// TIA Portal project "Banda_Asamblare" (V15.1)

(* hardware
DEVICE "S71500/ET200MP station_1"  S7-1500 station
   slot 0: "Rail_0"  Rack  6ES7 590-1***0-0AA0
   slot 1: "PLC_1"  CPU 1513-1 PN  6ES7 513-1AL02-0AB0  V2.6
      slot 3: "CPU display_1"  6ES7591-1AA00-0AA0
DEVICE "HMI_1"  KTP900 Basic PN
   slot 0: "HMI_1"  KTP900 Basic PN  6AV2 123-2JB03-0AX0  15.1.0.0
   slot 1: "HMI_RT_1"  KTP900 Basic PN  6AV2 123-2JB03-0AX0  15.1.0.0
   slot 5: "HMI_1.IE_CP_1"  PROFINET Interface  15.0.1.0
      slot 1: "PROFINET Interface_1"  PROFINET Interface
         slot 1: "Port_1"  Port
*)

// ===== PLC "PLC_1"  CPU 1513-1 PN =====

VAR_GLOBAL   // PLC tag table "Default tag table"
   "Clock_Byte" AT %MB0 : Byte;
   "Clock_10Hz" AT %M0.0 : Bool;
   "Clock_5Hz" AT %M0.1 : Bool;
   "Clock_2.5Hz" AT %M0.2 : Bool;
   "Clock_2Hz" AT %M0.3 : Bool;
   "Clock_1.25Hz" AT %M0.4 : Bool;
   "Clock_1Hz" AT %M0.5 : Bool;
   "Clock_0.625Hz" AT %M0.6 : Bool;
   "Clock_0.5Hz" AT %M0.7 : Bool;
END_VAR

DATA_BLOCK "Banda1_Avarii"   // DB1
{ S7_Optimized_Access := 'TRUE' }
VERSION : 0.1
   VAR
      avarie_start : Bool;
      avarie_cuptor : Bool;
      avarie_aplatizor : Bool;
      avarie_forme : Bool;
      avarie_taiere : Bool;
      avarie_curatare : Bool;
   END_VAR
BEGIN
END_DATA_BLOCK

DATA_BLOCK "Banda1_Butoane"   // DB2
{ S7_Optimized_Access := 'TRUE' }
VERSION : 0.1
   VAR
      btn_stop : Bool;
      btn_start : Bool;
      "reset avarii" : Bool;
   END_VAR
BEGIN
END_DATA_BLOCK

DATA_BLOCK "Banda_Principala_Avarii"   // DB3
{ S7_Optimized_Access := 'TRUE' }
VERSION : 0.1
   VAR
      esd : Bool;
      btn_esd : Bool;
      reset_est : Bool;
      btn_reset_avarii : Bool;
      avarii_generale : Bool;
      avarie_piesa1 : Bool;
      avarie_piesa2 : Bool;
      avarie_piesa3 : Bool;
   END_VAR
BEGIN
END_DATA_BLOCK

DATA_BLOCK "Banda1_Mecanisme"   // DB4
{ S7_Optimized_Access := 'TRUE' }
VERSION : 0.1
   VAR
      cuptor : Bool;
      temperatura_cuptor : Real;
      "temperatura dorita la cuptor" : Real;
      aplatizor : Bool;
      forma : UInt;
      ajuns_la_forma1 : Bool;
      ajuns_la_forma2 : Bool;
      ajuns_la_forma3 : Bool;
      taiere1 : Bool;
      taiere2 : Bool;
      taiere3 : Bool;
      curatare1 : Bool;
      curatare2 : Bool;
      curatare3 : Bool;
   END_VAR
BEGIN
END_DATA_BLOCK

DATA_BLOCK "Banda2_Butoane"   // DB5
{ S7_Optimized_Access := 'TRUE' }
VERSION : 0.1
   VAR
      btn_stop : Bool;
      btn_start : Bool;
      "reset avarii" : Bool;
   END_VAR
BEGIN
END_DATA_BLOCK

DATA_BLOCK "Banda1_DB"   // DB6
{ S7_Optimized_Access := 'TRUE' }
VERSION : 0.1
// stored: InstanceOfName Banda1
"Banda1"
BEGIN
END_DATA_BLOCK

DATA_BLOCK "Banda3_DB"   // DB7
{ S7_Optimized_Access := 'TRUE' }
VERSION : 0.1
// stored: InstanceOfName Banda1
"Banda1"
BEGIN
END_DATA_BLOCK

DATA_BLOCK "Banda2_DB"   // DB8
{ S7_Optimized_Access := 'TRUE' }
VERSION : 0.1
// stored: InstanceOfName Banda1
"Banda1"
BEGIN
END_DATA_BLOCK

DATA_BLOCK "Banda1_Alarme"   // DB9
{ S7_Optimized_Access := 'TRUE' }
VERSION : 0.1
   VAR
      alarme_gather : Word;
      alarme_vect : Array[0..15] of Bool;
   END_VAR
BEGIN
END_DATA_BLOCK

DATA_BLOCK "Banda2_Alarme"   // DB11
{ S7_Optimized_Access := 'TRUE' }
VERSION : 0.1
   VAR
      alarme_gather : Word;
      alarme_vect : Array[0..15] of Bool;
   END_VAR
BEGIN
END_DATA_BLOCK

DATA_BLOCK "Banda3_Alarme"   // DB12
{ S7_Optimized_Access := 'TRUE' }
VERSION : 0.1
   VAR
      alarme_gather : Word;
      alarme_vect : Array[0..15] of Bool;
   END_VAR
BEGIN
END_DATA_BLOCK

DATA_BLOCK "Banda2_Avarii"   // DB14
{ S7_Optimized_Access := 'TRUE' }
VERSION : 0.1
   VAR
      avarie_start : Bool;
      avarie_cuptor : Bool;
      avarie_aplatizor : Bool;
      avarie_forme : Bool;
      avarie_taiere : Bool;
      avarie_curatare : Bool;
   END_VAR
BEGIN
END_DATA_BLOCK

DATA_BLOCK "Banda3_Avarii"   // DB15
{ S7_Optimized_Access := 'TRUE' }
VERSION : 0.1
   VAR
      avarie_start : Bool;
      avarie_cuptor : Bool;
      avarie_aplatizor : Bool;
      avarie_forme : Bool;
      avarie_taiere : Bool;
      avarie_curatare : Bool;
   END_VAR
BEGIN
END_DATA_BLOCK

DATA_BLOCK "Containere"   // DB16
{ S7_Optimized_Access := 'TRUE' }
VERSION : 0.1
   VAR
      container1_plin : Bool;
      container2_plin : Bool;
      container3_plin : Bool;
      container_plin_general : Bool;
      limite_containere : Bool;
      golire_c1 : Bool;
      golire_c2 : Bool;
      golire_c3 : Bool;
      container_f1 : UInt;
      container_f2 : UInt;
      container_f3 : UInt;
      limita_c1 : UInt;
      limita_c2 : UInt;
      limita_c3 : UInt;
      container_plin : Bool;
      c1_plin : Bool;
      c2_plin : Bool;
      c3_plin : Bool;
      container_final : UInt;
      limita_container_final : UInt;
      cf_plin : Bool;
      golire_cf : Bool;
      container_f1_b1 : UInt;
      container_f1_b2 : UInt;
      container_f1_b3 : UInt;
      container_f2_b1 : UInt;
      container_f2_b2 : UInt;
      container_f2_b3 : UInt;
      container_f3_b1 : UInt;
      container_f3_b2 : UInt;
      container_f3_b3 : UInt;
      container_final_1 : UInt;
      container_final_2 : UInt;
      container_final_3 : UInt;
   END_VAR
BEGIN
END_DATA_BLOCK

DATA_BLOCK "Banda3_Butoane"   // DB17
{ S7_Optimized_Access := 'TRUE' }
VERSION : 0.1
   VAR
      btn_stop : Bool;
      btn_start : Bool;
      "reset avarii" : Bool;
   END_VAR
BEGIN
END_DATA_BLOCK

DATA_BLOCK "Banda2_Mecanisme"   // DB18
{ S7_Optimized_Access := 'TRUE' }
VERSION : 0.1
   VAR
      cuptor : Bool;
      temperatura_cuptor : Real;
      "temperatura dorita la cuptor" : Real;
      aplatizor : Bool;
      forma : UInt;
      ajuns_la_forma1 : Bool;
      ajuns_la_forma2 : Bool;
      ajuns_la_forma3 : Bool;
      taiere1 : Bool;
      taiere2 : Bool;
      taiere3 : Bool;
      curatare1 : Bool;
      curatare2 : Bool;
      curatare3 : Bool;
   END_VAR
BEGIN
END_DATA_BLOCK

DATA_BLOCK "Banda3_Mecanisme"   // DB19
{ S7_Optimized_Access := 'TRUE' }
VERSION : 0.1
   VAR
      cuptor : Bool;
      temperatura_cuptor : Real;
      "temperatura dorita la cuptor" : Real;
      aplatizor : Bool;
      forma : UInt;
      ajuns_la_forma1 : Bool;
      ajuns_la_forma2 : Bool;
      ajuns_la_forma3 : Bool;
      taiere1 : Bool;
      taiere2 : Bool;
      taiere3 : Bool;
      curatare1 : Bool;
      curatare2 : Bool;
      curatare3 : Bool;
   END_VAR
BEGIN
END_DATA_BLOCK

DATA_BLOCK "Banda_Principala_Alarme"   // DB20
{ S7_Optimized_Access := 'TRUE' }
VERSION : 0.1
   VAR
      alarme_gather : Word;
      alarme_vector : Array[0..15] of Bool;
   END_VAR
BEGIN
END_DATA_BLOCK

DATA_BLOCK "Containere_Alarme"   // DB24
{ S7_Optimized_Access := 'TRUE' }
VERSION : 0.1
   VAR
      alarme_gather : Word;
      alarme_vector : Array[0..15] of Bool;
   END_VAR
BEGIN
END_DATA_BLOCK

DATA_BLOCK "Banda_Principala_Butoane"   // DB25
{ S7_Optimized_Access := 'TRUE' }
VERSION : 0.1
   VAR
      start_btn : Bool;
      stop_btn : Bool;
      pornire : Bool;
      pune_1 : Bool;
      pune_2 : Bool;
      pune_3 : Bool;
      trece_1 : Bool;
      trece_2 : Bool;
      trece_3 : Bool;
      resetare : Bool;
   END_VAR
BEGIN
END_DATA_BLOCK

DATA_BLOCK "Banda_Principala_Comenzi_DB"   // DB28
{ S7_Optimized_Access := 'TRUE' }
VERSION : 0.1
// stored: InstanceOfName Banda_Principala_Comenzi
"Banda_Principala_Comenzi"
BEGIN
END_DATA_BLOCK

DATA_BLOCK "Banda_Principala_Simulare_DB"   // DB29
{ S7_Optimized_Access := 'TRUE' }
VERSION : 0.1
// stored: InstanceOfName Banda_Principala_Simulare
"Banda_Principala_Simulare"
BEGIN
END_DATA_BLOCK

// folder: System blocks/Program resources

DATA_BLOCK "reset_buton_oprite_banda_principala"   // DB10
{ S7_Optimized_Access := 'TRUE' }
AUTHOR : Simatic
FAMILY : IEC
NAME : IEC_TMR
VERSION : 1.0
// stored: InstanceOfName IEC_TIMER
"IEC_TIMER"
BEGIN
END_DATA_BLOCK

DATA_BLOCK "reset_esd_timer"   // DB26
{ S7_Optimized_Access := 'TRUE' }
AUTHOR : Simatic
FAMILY : IEC
NAME : IEC_TMR
VERSION : 1.0
// stored: InstanceOfName IEC_TIMER
"IEC_TIMER"
BEGIN
END_DATA_BLOCK

// folder: (top level)

FUNCTION_BLOCK "Simulare1"   // FB1, LAD
{ S7_Optimized_Access := 'TRUE' }
VERSION : 0.1
   VAR_INPUT
      btn_pornire : Bool;
      b1_plecat : Bool;
      b2_plecat : Bool;
      b3_plecat : Bool;
      b41_plecat : Bool;
      b42_plecat : Bool;
      b43_plecat : Bool;
      b51_plecat : Bool;
      b52_plecat : Bool;
      b53_plecat : Bool;
      b61_plecat : Bool;
      b62_plecat : Bool;
      b63_plecat : Bool;
      cond_cuptor : Bool;
      forma : UInt;
      trecere_banda_mare1 : Bool;
      trecere_banda_mare2 : Bool;
      trecere_banda_mare3 : Bool;
   END_VAR
   VAR_OUTPUT
      cuptor_pornit : Bool;
      aplatizor_pornit : Bool;
      forma1 : Bool;
      forma2 : Bool;
      forma3 : Bool;
      taiere1 : Bool;
      taiere2 : Bool;
      taiere3 : Bool;
      curatare1 : Bool;
      curatare2 : Bool;
      curatare3 : Bool;
      container1 : UInt;
      container2 : UInt;
      container3 : UInt;
      servo : UInt;
   END_VAR
   VAR_IN_OUT
      pune_material : Bool;
      temp_cuptor : Real;
      golire_c1 : Bool;
      golire_c2 : Bool;
      golire_c3 : Bool;
   END_VAR
   VAR
      re1 : Bool;
      re2 : Bool;
      re3 : Bool;
      re4 : Bool;
      re5 : Bool;
      re6 : Bool;
      re7 : Bool;
      re8 : Bool;
      "timer reset punere material" : TON_TIME;
      mentinere_timer_material : Bool;
      timer_aplatizare : TON_TIME;
      "tiimer forma" : TON_TIME;
      "timer taiere1" : TON_TIME;
      "timer taiere2" : TON_TIME;
      "timer taiere3" : TON_TIME;
      "timer curatare1" : TON_TIME;
      "timer curatare 2" : TON_TIME;
      "timer curatare 3" : TON_TIME;
      reset_golire1 : TON_TIME;
      reset_golire2 : TON_TIME;
      reset_golire3 : TON_TIME;
      scazut1 : Bool;
      scazut2 : Bool;
      scazut3 : Bool;
   END_VAR
   VAR_TEMP   // added for the SCL form of the ladder/FBD networks
      _w1 : Bool;
      _w2 : Bool;
      _w3 : Bool;
   END_VAR
BEGIN

REGION Network 1: pune un block de material pe banda
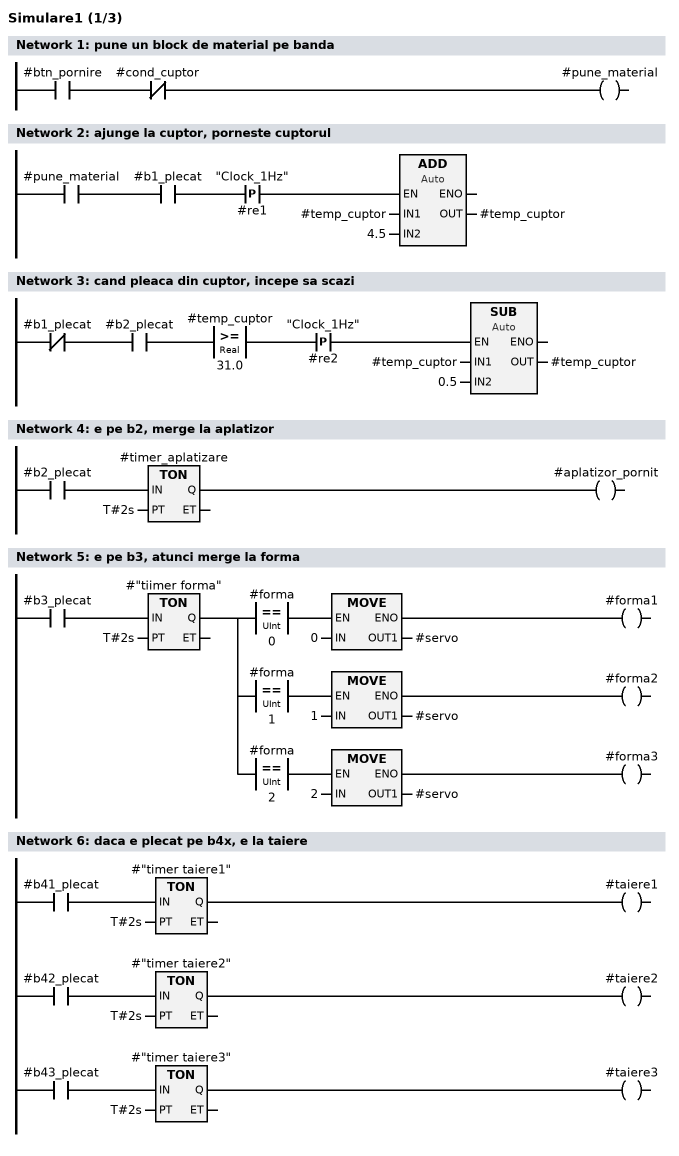
   RUNG wire#powerrail
      Contact( #btn_pornire )
      I_Contact( #cond_cuptor )
      Coil( #pune_material )
   END_RUNG
   // the same network as SCL:
   #pune_material := #btn_pornire AND NOT #cond_cuptor;
END_REGION

REGION Network 2: ajunge la cuptor, porneste cuptorul
   RUNG wire#powerrail
      Contact( #pune_material )
      Contact( #b1_plecat )
      P_Contact(operand := "Clock_1Hz", bit := #re1)
      Add(in1 := #temp_cuptor, in2 := 4.5, out => #temp_cuptor)
   END_RUNG
   // the same network as SCL:
   #_w1 := #pune_material AND #b1_plecat AND "Clock_1Hz" AND NOT #re1;   // rising edge of "Clock_1Hz"
   #re1 := "Clock_1Hz";
   IF #_w1 THEN #temp_cuptor := #temp_cuptor + 4.5; END_IF;
END_REGION

REGION Network 3: cand pleaca din cuptor, incepe sa scazi
   RUNG wire#powerrail
      I_Contact( #b1_plecat )
      Contact( #b2_plecat )
      { S7_Templates := "SrcType := Real" } GE_Contact(in1 := #temp_cuptor, in2 := 31.0)
      P_Contact(operand := "Clock_1Hz", bit := #re2)
      Sub(in1 := #temp_cuptor, in2 := 0.5, out => #temp_cuptor)
   END_RUNG
   // the same network as SCL:
   #_w1 := NOT #b1_plecat AND #b2_plecat AND (#temp_cuptor >= 31.0) AND "Clock_1Hz" AND NOT #re2;   // rising edge of "Clock_1Hz"
   #re2 := "Clock_1Hz";
   IF #_w1 THEN #temp_cuptor := #temp_cuptor - 0.5; END_IF;
END_REGION

REGION Network 4: e pe b2, merge la aplatizor
   #timer_aplatizare(IN := #b2_plecat, PT := T#2s);   // TON
   #aplatizor_pornit := #timer_aplatizare.Q;
END_REGION

REGION Network 5: e pe b3, atunci merge la forma
   #"tiimer forma"(IN := #b3_plecat, PT := T#2s);   // TON
   #_w1 := #"tiimer forma".Q AND (#forma = 0);
   IF #_w1 THEN #servo := 0; END_IF;
   #forma1 := #_w1;
   #_w2 := #"tiimer forma".Q AND (#forma = 1);
   IF #_w2 THEN #servo := 1; END_IF;
   #forma2 := #_w2;
   #_w3 := #"tiimer forma".Q AND (#forma = 2);
   IF #_w3 THEN #servo := 2; END_IF;
   #forma3 := #_w3;
END_REGION

REGION Network 6: daca e plecat pe b4x, e la taiere
   #"timer taiere1"(IN := #b41_plecat, PT := T#2s);   // TON
   #taiere1 := #"timer taiere1".Q;
   #"timer taiere2"(IN := #b42_plecat, PT := T#2s);   // TON
   #taiere2 := #"timer taiere2".Q;
   #"timer taiere3"(IN := #b43_plecat, PT := T#2s);   // TON
   #taiere3 := #"timer taiere3".Q;
END_REGION

REGION Network 7: daca e pe banda b5x, sa dea drumul la curatari
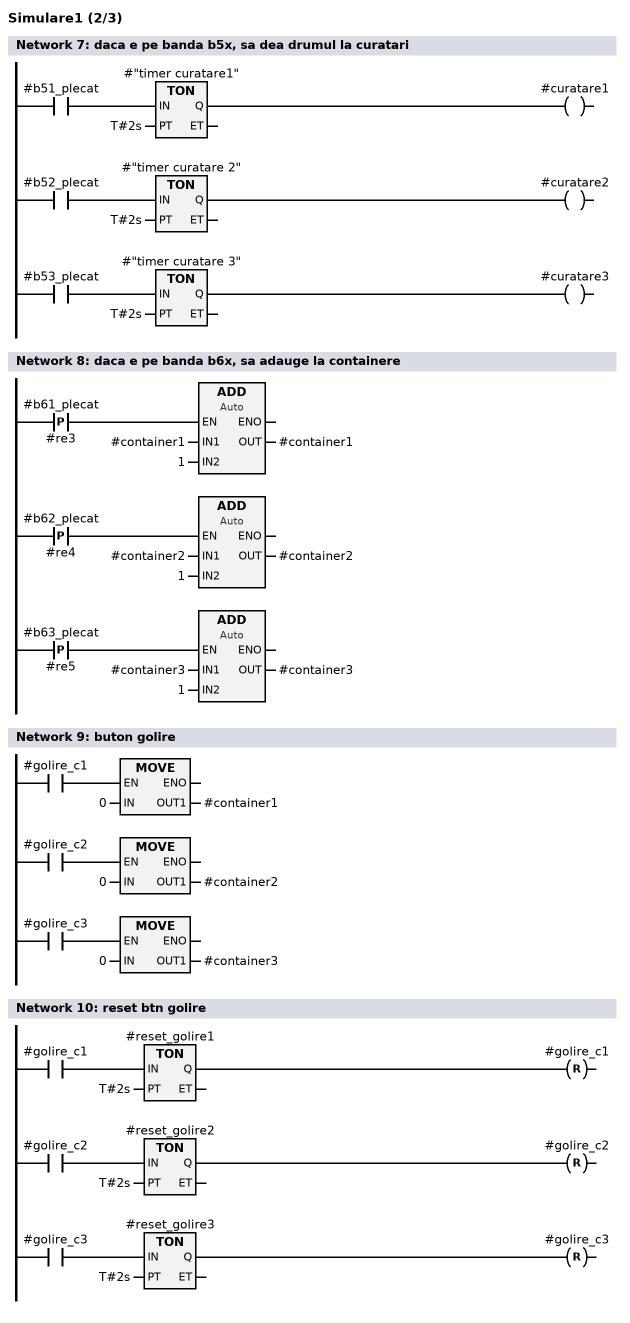
   #"timer curatare1"(IN := #b51_plecat, PT := T#2s);   // TON
   #curatare1 := #"timer curatare1".Q;
   #"timer curatare 2"(IN := #b52_plecat, PT := T#2s);   // TON
   #curatare2 := #"timer curatare 2".Q;
   #"timer curatare 3"(IN := #b53_plecat, PT := T#2s);   // TON
   #curatare3 := #"timer curatare 3".Q;
END_REGION

REGION Network 8: daca e pe banda b6x, sa adauge la containere
   RUNG wire#powerrail
      P_Contact(operand := #b61_plecat, bit := #re3)
      Add(in1 := #container1, in2 := 1, out => #container1)
   END_RUNG
   RUNG wire#powerrail
      P_Contact(operand := #b62_plecat, bit := #re4)
      Add(in1 := #container2, in2 := 1, out => #container2)
   END_RUNG
   RUNG wire#powerrail
      P_Contact(operand := #b63_plecat, bit := #re5)
      Add(in1 := #container3, in2 := 1, out => #container3)
   END_RUNG
   // the same network as SCL:
   #_w1 := #b61_plecat AND NOT #re3;   // rising edge of #b61_plecat
   #re3 := #b61_plecat;
   IF #_w1 THEN #container1 := #container1 + 1; END_IF;
   #_w2 := #b62_plecat AND NOT #re4;   // rising edge of #b62_plecat
   #re4 := #b62_plecat;
   IF #_w2 THEN #container2 := #container2 + 1; END_IF;
   #_w3 := #b63_plecat AND NOT #re5;   // rising edge of #b63_plecat
   #re5 := #b63_plecat;
   IF #_w3 THEN #container3 := #container3 + 1; END_IF;
END_REGION

REGION Network 9: buton golire
   RUNG wire#powerrail
      Contact( #golire_c1 )
      Move(in := 0, out1 => #container1)
   END_RUNG
   RUNG wire#powerrail
      Contact( #golire_c2 )
      Move(in := 0, out1 => #container2)
   END_RUNG
   RUNG wire#powerrail
      Contact( #golire_c3 )
      Move(in := 0, out1 => #container3)
   END_RUNG
   // the same network as SCL:
   IF #golire_c1 THEN #container1 := 0; END_IF;
   IF #golire_c2 THEN #container2 := 0; END_IF;
   IF #golire_c3 THEN #container3 := 0; END_IF;
END_REGION

REGION Network 10: reset btn golire
   #reset_golire1(IN := #golire_c1, PT := T#2s);   // TON
   IF #reset_golire1.Q THEN #golire_c1 := FALSE; END_IF;
   #reset_golire2(IN := #golire_c2, PT := T#2s);   // TON
   IF #reset_golire2.Q THEN #golire_c2 := FALSE; END_IF;
   #reset_golire3(IN := #golire_c3, PT := T#2s);   // TON
   IF #reset_golire3.Q THEN #golire_c3 := FALSE; END_IF;
END_REGION

REGION Network 11: daca avem treceri de pe banda mare, scadem valoarea din containere
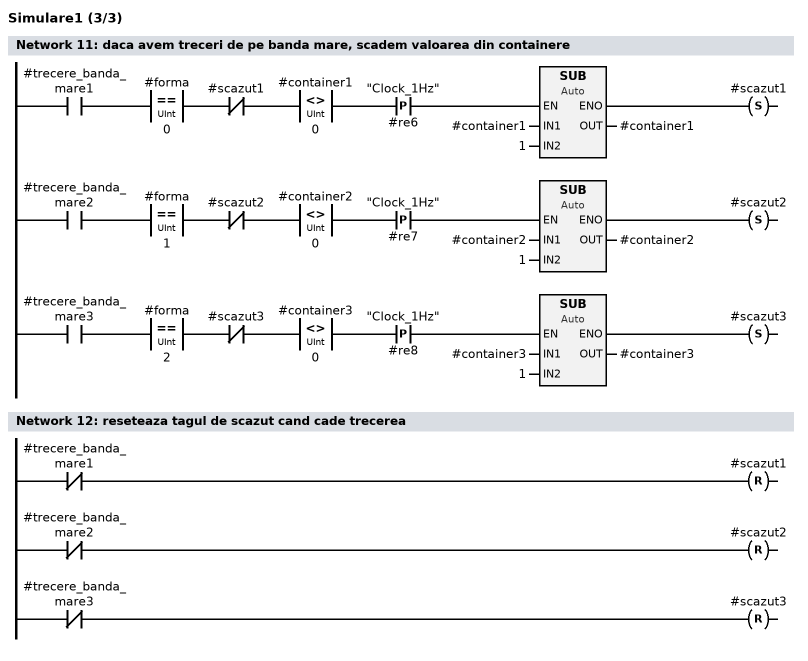
   RUNG wire#powerrail
      Contact( #trecere_banda_mare1 )
      { S7_Templates := "SrcType := UInt" } EQ_Contact(in1 := #forma, in2 := 0)
      I_Contact( #scazut1 )
      { S7_Templates := "SrcType := UInt" } NE_Contact(in1 := #container1, in2 := 0)
      P_Contact(operand := "Clock_1Hz", bit := #re6)
      Sub(in1 := #container1, in2 := 1, out => #container1)
      S_Coil( #scazut1 )
   END_RUNG
   RUNG wire#powerrail
      Contact( #trecere_banda_mare2 )
      { S7_Templates := "SrcType := UInt" } EQ_Contact(in1 := #forma, in2 := 1)
      I_Contact( #scazut2 )
      { S7_Templates := "SrcType := UInt" } NE_Contact(in1 := #container2, in2 := 0)
      P_Contact(operand := "Clock_1Hz", bit := #re7)
      Sub(in1 := #container2, in2 := 1, out => #container2)
      S_Coil( #scazut2 )
   END_RUNG
   RUNG wire#powerrail
      Contact( #trecere_banda_mare3 )
      { S7_Templates := "SrcType := UInt" } EQ_Contact(in1 := #forma, in2 := 2)
      I_Contact( #scazut3 )
      { S7_Templates := "SrcType := UInt" } NE_Contact(in1 := #container3, in2 := 0)
      P_Contact(operand := "Clock_1Hz", bit := #re8)
      Sub(in1 := #container3, in2 := 1, out => #container3)
      S_Coil( #scazut3 )
   END_RUNG
   // the same network as SCL:
   #_w1 := #trecere_banda_mare1 AND (#forma = 0) AND NOT #scazut1 AND (#container1 <> 0) AND "Clock_1Hz" AND NOT #re6;   // rising edge of "Clock_1Hz"
   #re6 := "Clock_1Hz";
   IF #_w1 THEN
       #container1 := #container1 - 1;
       #scazut1 := TRUE;
   END_IF;
   #_w2 := #trecere_banda_mare2 AND (#forma = 1) AND NOT #scazut2 AND (#container2 <> 0) AND "Clock_1Hz" AND NOT #re7;   // rising edge of "Clock_1Hz"
   #re7 := "Clock_1Hz";
   IF #_w2 THEN
       #container2 := #container2 - 1;
       #scazut2 := TRUE;
   END_IF;
   #_w3 := #trecere_banda_mare3 AND (#forma = 2) AND NOT #scazut3 AND (#container3 <> 0) AND "Clock_1Hz" AND NOT #re8;   // rising edge of "Clock_1Hz"
   #re8 := "Clock_1Hz";
   IF #_w3 THEN
       #container3 := #container3 - 1;
       #scazut3 := TRUE;
   END_IF;
END_REGION

REGION Network 12: reseteaza tagul de scazut cand cade trecerea
   RUNG wire#powerrail
      I_Contact( #trecere_banda_mare1 )
      R_Coil( #scazut1 )
   END_RUNG
   RUNG wire#powerrail
      I_Contact( #trecere_banda_mare2 )
      R_Coil( #scazut2 )
   END_RUNG
   RUNG wire#powerrail
      I_Contact( #trecere_banda_mare3 )
      R_Coil( #scazut3 )
   END_RUNG
   // the same network as SCL:
   IF NOT #trecere_banda_mare1 THEN #scazut1 := FALSE; END_IF;
   IF NOT #trecere_banda_mare2 THEN #scazut2 := FALSE; END_IF;
   IF NOT #trecere_banda_mare3 THEN #scazut3 := FALSE; END_IF;
END_REGION
END_FUNCTION_BLOCK

FUNCTION_BLOCK "Comenzi1"   // FB2, LAD
{ S7_Optimized_Access := 'TRUE' }
VERSION : 0.1
   VAR_INPUT
      temp_cuptor : Real;
      temp_dorita : Real;
      pune_material : Bool;
      aplatizor_pornit : Bool;
      forma1 : Bool;
      forma2 : Bool;
      forma3 : Bool;
      taiere1 : Bool;
      taiere2 : Bool;
      taiere3 : Bool;
      curatare1 : Bool;
      curatare2 : Bool;
      curatare3 : Bool;
   END_VAR
   VAR_OUTPUT
      b1_plecat : Bool;
      b2_plecat : Bool;
      b3_plecat : Bool;
      b41_plecat : Bool;
      b42_plecat : Bool;
      b43_plecat : Bool;
      b51_plecat : Bool;
      b52_plecat : Bool;
      b53_plecat : Bool;
      b61_plecat : Bool;
      b62_plecat : Bool;
      b63_plecat : Bool;
      cond_cuptor : Bool;
   END_VAR
   VAR
      "timer plecare b1" : TON_TIME;
      incc : Int;
      edg : Bool;
   END_VAR
BEGIN

REGION Network 1: pleaca spre cuptor
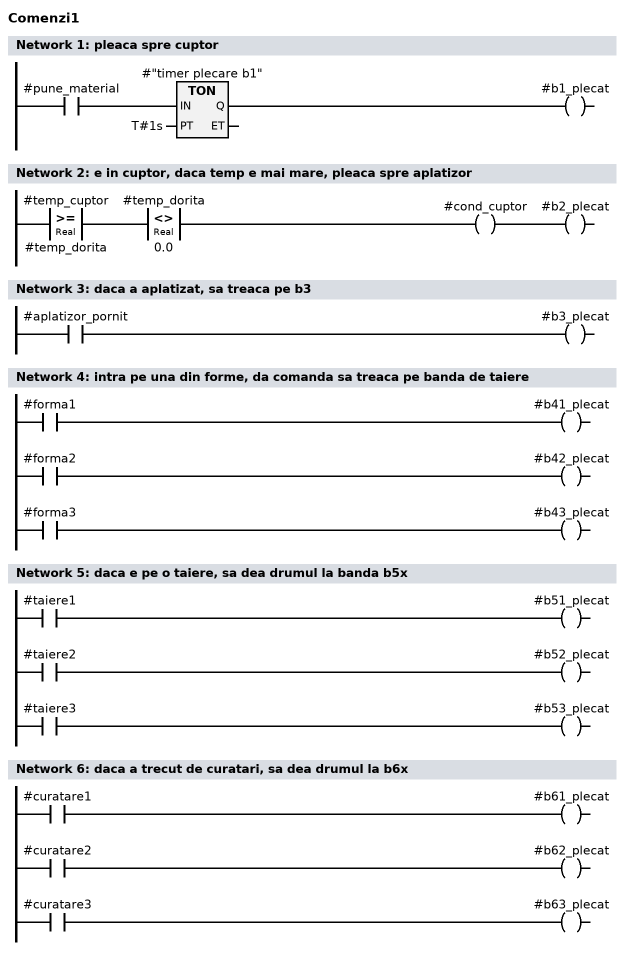
   #"timer plecare b1"(IN := #pune_material, PT := T#1s);   // TON
   #b1_plecat := #"timer plecare b1".Q;
END_REGION

REGION Network 2: e in cuptor, daca temp e mai mare, pleaca spre aplatizor
   RUNG wire#powerrail
      { S7_Templates := "SrcType := Real" } GE_Contact(in1 := #temp_cuptor, in2 := #temp_dorita)
      { S7_Templates := "SrcType := Real" } NE_Contact(in1 := #temp_dorita, in2 := 0.0)
      Coil( #cond_cuptor )
      Coil( #b2_plecat )
   END_RUNG
   // the same network as SCL:
   #cond_cuptor := (#temp_cuptor >= #temp_dorita) AND (#temp_dorita <> 0.0);
   #b2_plecat := #cond_cuptor;
END_REGION

REGION Network 3: daca a aplatizat, sa treaca pe b3
   RUNG wire#powerrail
      Contact( #aplatizor_pornit )
      Coil( #b3_plecat )
   END_RUNG
   // the same network as SCL:
   #b3_plecat := #aplatizor_pornit;
END_REGION

REGION Network 4: intra pe una din forme, da comanda sa treaca pe banda de taiere
   RUNG wire#powerrail
      Contact( #forma1 )
      Coil( #b41_plecat )
   END_RUNG
   RUNG wire#powerrail
      Contact( #forma2 )
      Coil( #b42_plecat )
   END_RUNG
   RUNG wire#powerrail
      Contact( #forma3 )
      Coil( #b43_plecat )
   END_RUNG
   // the same network as SCL:
   #b41_plecat := #forma1;
   #b42_plecat := #forma2;
   #b43_plecat := #forma3;
END_REGION

REGION Network 5: daca e pe o taiere, sa dea drumul la banda b5x
   RUNG wire#powerrail
      Contact( #taiere1 )
      Coil( #b51_plecat )
   END_RUNG
   RUNG wire#powerrail
      Contact( #taiere2 )
      Coil( #b52_plecat )
   END_RUNG
   RUNG wire#powerrail
      Contact( #taiere3 )
      Coil( #b53_plecat )
   END_RUNG
   // the same network as SCL:
   #b51_plecat := #taiere1;
   #b52_plecat := #taiere2;
   #b53_plecat := #taiere3;
END_REGION

REGION Network 6: daca a trecut de curatari, sa dea drumul la b6x
   RUNG wire#powerrail
      Contact( #curatare1 )
      Coil( #b61_plecat )
   END_RUNG
   RUNG wire#powerrail
      Contact( #curatare2 )
      Coil( #b62_plecat )
   END_RUNG
   RUNG wire#powerrail
      Contact( #curatare3 )
      Coil( #b63_plecat )
   END_RUNG
   // the same network as SCL:
   #b61_plecat := #curatare1;
   #b62_plecat := #curatare2;
   #b63_plecat := #curatare3;
END_REGION
END_FUNCTION_BLOCK

FUNCTION_BLOCK "Banda1"   // FB3, LAD
{ S7_Optimized_Access := 'TRUE' }
VERSION : 0.1
   VAR_INPUT
      temperatura_dorita : Real := 0.0;
      forma : UInt := 0;
      limita_container1 : UInt;
      limita_container2 : UInt;
      limita_container3 : UInt;
      container_plin : Bool;
      trecere_banda_mare1 : Bool;
      trecere_banda_mare2 : Bool;
      trecere_banda_mare3 : Bool;
   END_VAR
   VAR_OUTPUT
      container1 : UInt;
      container2 : UInt;
      container3 : UInt;
      cuptor : Bool;
      aplatizor : Bool;
      ajuns_forma1 : Bool;
      ajuns_forma2 : Bool;
      ajuns_forma3 : Bool;
      taiere1 : Bool;
      taiere2 : Bool;
      taiere3 : Bool;
      curatare1 : Bool;
      curatare2 : Bool;
      curatare3 : Bool;
      alarme_gather : Word;
      alarme_vect : Array[0..15] of Bool;
   END_VAR
   VAR_IN_OUT
      stop : Bool;
      start : Bool;
      golire_c1 : Bool;
      golire_c2 : Bool;
      golire_c3 : Bool;
      btn_reset_avarii : Bool;
      avarie_start : Bool;
      avarie_cuptor : Bool;
      avarie_aplatizor : Bool;
      avarie_forma : Bool;
      avarie_taiere : Bool;
      avarie_curatare : Bool;
      temperatura_cuptor : Real;
      esd : Bool;
   END_VAR
   VAR
      limite_containere : Bool;
      Avarii_generale : Bool;
      pornire : Bool;
      punere_block : Bool;
      plecat_b1 : Bool;
      plecat_b2 : Bool;
      plecat_b3 : Bool;
      plecat_b41 : Bool;
      plecat_b42 : Bool;
      plecat_b43 : Bool;
      plecar_b51 : Bool;
      plecar_b52 : Bool;
      plecar_b53 : Bool;
      plecat_b61 : Bool;
      plecat_b62 : Bool;
      plecat_b63 : Bool;
      cond_cuptor : Bool;
      servo : UInt;
      reset_esd_timer : TON_TIME;
      plin_container1 : Bool;
      plin_container2 : Bool;
      plin_container3 : Bool;
      reset_btn_stop : TON_TIME;
      Simulare1_Instance : "Simulare1";
      Comenzi1_Instance : "Comenzi1";
   END_VAR
BEGIN

REGION Network 1: buton start
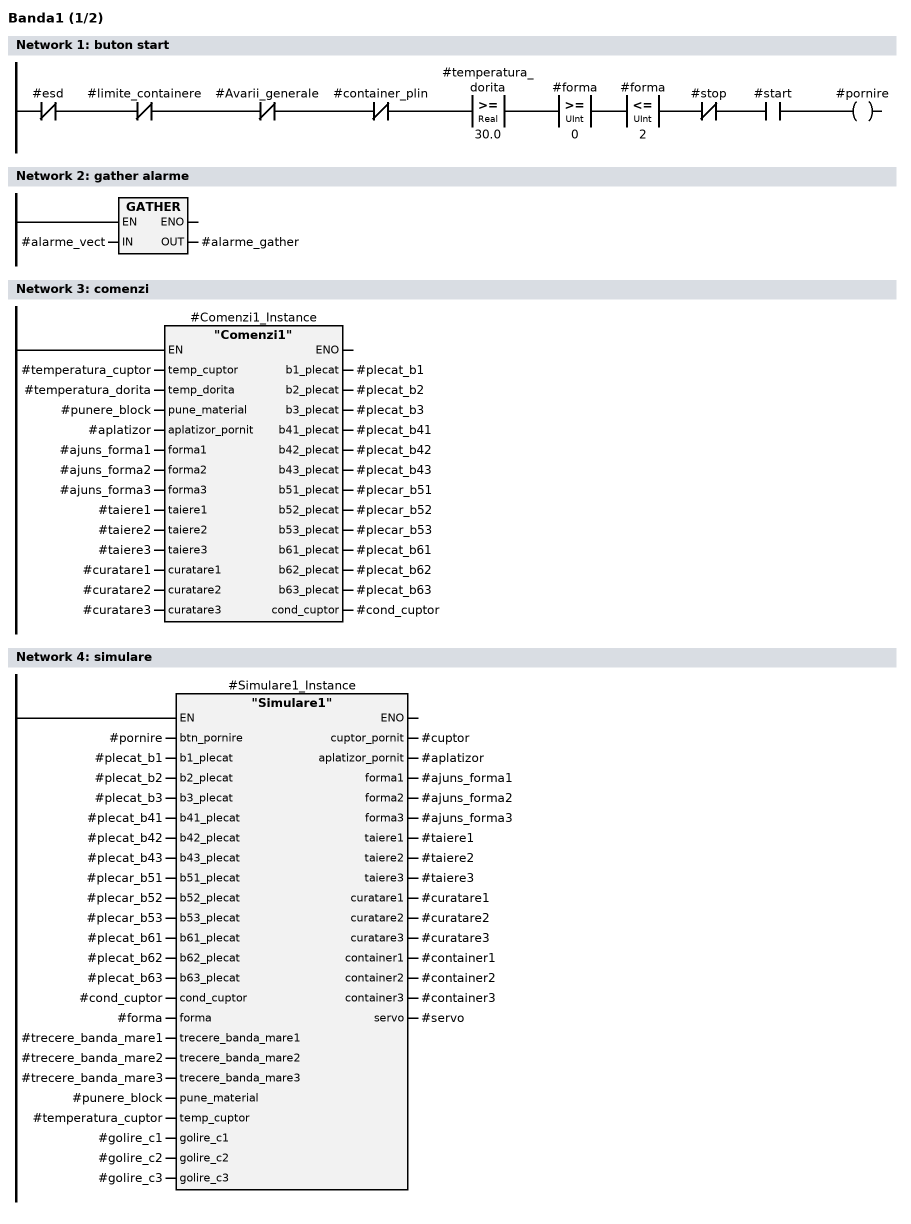
   RUNG wire#powerrail
      I_Contact( #esd )
      I_Contact( #limite_containere )
      I_Contact( #Avarii_generale )
      I_Contact( #container_plin )
      { S7_Templates := "SrcType := Real" } GE_Contact(in1 := #temperatura_dorita, in2 := 30.0)
      { S7_Templates := "SrcType := UInt" } GE_Contact(in1 := #forma, in2 := 0)
      { S7_Templates := "SrcType := UInt" } LE_Contact(in1 := #forma, in2 := 2)
      I_Contact( #stop )
      Contact( #start )
      Coil( #pornire )
   END_RUNG
   // the same network as SCL:
   #pornire := NOT #esd AND NOT #limite_containere AND NOT #Avarii_generale AND NOT #container_plin AND (#temperatura_dorita >= 30.0) AND (#forma >= 0) AND (#forma <= 2) AND NOT #stop AND #start;
END_REGION

REGION Network 2: gather alarme
   GATHER(IN := #alarme_vect, OUT => #alarme_gather);
END_REGION

REGION Network 3: comenzi
   RUNG wire#powerrail
      #Comenzi1_Instance(temp_cuptor := #temperatura_cuptor, temp_dorita := #temperatura_dorita, pune_material := #punere_block, aplatizor_pornit := #aplatizor, forma1 := #ajuns_forma1, forma2 := #ajuns_forma2, forma3 := #ajuns_forma3, taiere1 := #taiere1, taiere2 := #taiere2, taiere3 := #taiere3, curatare1 := #curatare1, curatare2 := #curatare2, curatare3 := #curatare3, b1_plecat => #plecat_b1, b2_plecat => #plecat_b2, b3_plecat => #plecat_b3, b41_plecat => #plecat_b41, b42_plecat => #plecat_b42, b43_plecat => #plecat_b43, b51_plecat => #plecar_b51, b52_plecat => #plecar_b52, b53_plecat => #plecar_b53, b61_plecat => #plecat_b61, b62_plecat => #plecat_b62, b63_plecat => #plecat_b63, cond_cuptor => #cond_cuptor)
   END_RUNG
   // the same network as SCL:
   #Comenzi1_Instance(temp_cuptor := #temperatura_cuptor,   // "Comenzi1"
                      temp_dorita := #temperatura_dorita,
                      pune_material := #punere_block,
                      aplatizor_pornit := #aplatizor,
                      forma1 := #ajuns_forma1,
                      forma2 := #ajuns_forma2,
                      forma3 := #ajuns_forma3,
                      taiere1 := #taiere1,
                      taiere2 := #taiere2,
                      taiere3 := #taiere3,
                      curatare1 := #curatare1,
                      curatare2 := #curatare2,
                      curatare3 := #curatare3,
                      b1_plecat => #plecat_b1,
                      b2_plecat => #plecat_b2,
                      b3_plecat => #plecat_b3,
                      b41_plecat => #plecat_b41,
                      b42_plecat => #plecat_b42,
                      b43_plecat => #plecat_b43,
                      b51_plecat => #plecar_b51,
                      b52_plecat => #plecar_b52,
                      b53_plecat => #plecar_b53,
                      b61_plecat => #plecat_b61,
                      b62_plecat => #plecat_b62,
                      b63_plecat => #plecat_b63,
                      cond_cuptor => #cond_cuptor);
END_REGION

REGION Network 4: simulare
   RUNG wire#powerrail
      #Simulare1_Instance(btn_pornire := #pornire, b1_plecat := #plecat_b1, b2_plecat := #plecat_b2, b3_plecat := #plecat_b3, b41_plecat := #plecat_b41, b42_plecat := #plecat_b42, b43_plecat := #plecat_b43, b51_plecat := #plecar_b51, b52_plecat := #plecar_b52, b53_plecat := #plecar_b53, b61_plecat := #plecat_b61, b62_plecat := #plecat_b62, b63_plecat := #plecat_b63, cond_cuptor := #cond_cuptor, forma := #forma, trecere_banda_mare1 := #trecere_banda_mare1, trecere_banda_mare2 := #trecere_banda_mare2, trecere_banda_mare3 := #trecere_banda_mare3, pune_material := #punere_block, temp_cuptor := #temperatura_cuptor, golire_c1 := #golire_c1, golire_c2 := #golire_c2, golire_c3 := #golire_c3, cuptor_pornit => #cuptor, aplatizor_pornit => #aplatizor, forma1 => #ajuns_forma1, forma2 => #ajuns_forma2, forma3 => #ajuns_forma3, taiere1 => #taiere1, taiere2 => #taiere2, taiere3 => #taiere3, curatare1 => #curatare1, curatare2 => #curatare2, curatare3 => #curatare3, container1 => #container1, container2 => #container2, container3 => #container3, servo => #servo)
   END_RUNG
   // the same network as SCL:
   #Simulare1_Instance(btn_pornire := #pornire,   // "Simulare1"
                       b1_plecat := #plecat_b1,
                       b2_plecat := #plecat_b2,
                       b3_plecat := #plecat_b3,
                       b41_plecat := #plecat_b41,
                       b42_plecat := #plecat_b42,
                       b43_plecat := #plecat_b43,
                       b51_plecat := #plecar_b51,
                       b52_plecat := #plecar_b52,
                       b53_plecat := #plecar_b53,
                       b61_plecat := #plecat_b61,
                       b62_plecat := #plecat_b62,
                       b63_plecat := #plecat_b63,
                       cond_cuptor := #cond_cuptor,
                       forma := #forma,
                       trecere_banda_mare1 := #trecere_banda_mare1,
                       trecere_banda_mare2 := #trecere_banda_mare2,
                       trecere_banda_mare3 := #trecere_banda_mare3,
                       pune_material := #punere_block,
                       temp_cuptor := #temperatura_cuptor,
                       golire_c1 := #golire_c1,
                       golire_c2 := #golire_c2,
                       golire_c3 := #golire_c3,
                       cuptor_pornit => #cuptor,
                       aplatizor_pornit => #aplatizor,
                       forma1 => #ajuns_forma1,
                       forma2 => #ajuns_forma2,
                       forma3 => #ajuns_forma3,
                       taiere1 => #taiere1,
                       taiere2 => #taiere2,
                       taiere3 => #taiere3,
                       curatare1 => #curatare1,
                       curatare2 => #curatare2,
                       curatare3 => #curatare3,
                       container1 => #container1,
                       container2 => #container2,
                       container3 => #container3,
                       servo => #servo);
END_REGION

REGION Network 5: avarie generala
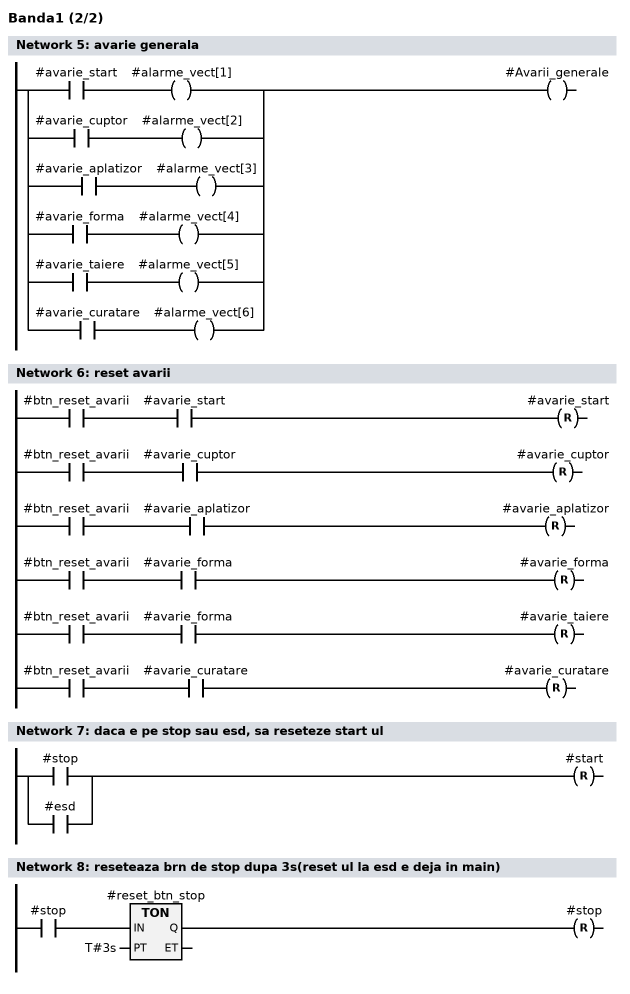
   RUNG wire#powerrail
      Contact( #avarie_start )
      Coil( #alarme_vect[1] )
      wire#w1
      Coil( #Avarii_generale )
   END_RUNG
   RUNG wire#powerrail
      Contact( #avarie_cuptor )
      Coil( #alarme_vect[2] )
   END_RUNG wire#w1
   RUNG wire#powerrail
      Contact( #avarie_aplatizor )
      Coil( #alarme_vect[3] )
   END_RUNG wire#w1
   RUNG wire#powerrail
      Contact( #avarie_forma )
      Coil( #alarme_vect[4] )
   END_RUNG wire#w1
   RUNG wire#powerrail
      Contact( #avarie_taiere )
      Coil( #alarme_vect[5] )
   END_RUNG wire#w1
   RUNG wire#powerrail
      Contact( #avarie_curatare )
      Coil( #alarme_vect[6] )
   END_RUNG wire#w1
   // the same network as SCL:
   #alarme_vect[1] := #avarie_start;
   #alarme_vect[2] := #avarie_cuptor;
   #alarme_vect[3] := #avarie_aplatizor;
   #alarme_vect[4] := #avarie_forma;
   #alarme_vect[5] := #avarie_taiere;
   #alarme_vect[6] := #avarie_curatare;
   #Avarii_generale := #avarie_start OR #avarie_cuptor OR #avarie_aplatizor OR #avarie_forma OR #avarie_taiere OR #avarie_curatare;
END_REGION

REGION Network 6: reset avarii
   RUNG wire#powerrail
      Contact( #btn_reset_avarii )
      Contact( #avarie_start )
      R_Coil( #avarie_start )
   END_RUNG
   RUNG wire#powerrail
      Contact( #btn_reset_avarii )
      Contact( #avarie_cuptor )
      R_Coil( #avarie_cuptor )
   END_RUNG
   RUNG wire#powerrail
      Contact( #btn_reset_avarii )
      Contact( #avarie_aplatizor )
      R_Coil( #avarie_aplatizor )
   END_RUNG
   RUNG wire#powerrail
      Contact( #btn_reset_avarii )
      Contact( #avarie_forma )
      R_Coil( #avarie_forma )
   END_RUNG
   RUNG wire#powerrail
      Contact( #btn_reset_avarii )
      Contact( #avarie_forma )
      R_Coil( #avarie_taiere )
   END_RUNG
   RUNG wire#powerrail
      Contact( #btn_reset_avarii )
      Contact( #avarie_curatare )
      R_Coil( #avarie_curatare )
   END_RUNG
   // the same network as SCL:
   IF #btn_reset_avarii AND #avarie_start THEN #avarie_start := FALSE; END_IF;
   IF #btn_reset_avarii AND #avarie_cuptor THEN #avarie_cuptor := FALSE; END_IF;
   IF #btn_reset_avarii AND #avarie_aplatizor THEN #avarie_aplatizor := FALSE; END_IF;
   IF #btn_reset_avarii AND #avarie_forma THEN #avarie_forma := FALSE; END_IF;
   IF #btn_reset_avarii AND #avarie_forma THEN #avarie_taiere := FALSE; END_IF;
   IF #btn_reset_avarii AND #avarie_curatare THEN #avarie_curatare := FALSE; END_IF;
END_REGION

REGION Network 7: daca e pe stop sau esd, sa reseteze start ul
   RUNG wire#powerrail
      Contact( #stop )
      wire#w1
      R_Coil( #start )
   END_RUNG
   RUNG wire#powerrail
      Contact( #esd )
   END_RUNG wire#w1
   // the same network as SCL:
   IF #stop OR #esd THEN #start := FALSE; END_IF;
END_REGION

REGION Network 8: reseteaza brn de stop dupa 3s(reset ul la esd e deja in main)
   #reset_btn_stop(IN := #stop, PT := T#3s);   // TON
   IF #reset_btn_stop.Q THEN #stop := FALSE; END_IF;
END_REGION
END_FUNCTION_BLOCK

FUNCTION_BLOCK "Banda_Principala_Comenzi"   // FB4, LAD
{ S7_Optimized_Access := 'TRUE' }
VERSION : 0.1
   VAR_INPUT
      pornire : Bool;
      trecut1 : Bool;
      trecut2 : Bool;
      resetare : Bool;
   END_VAR
   VAR_OUTPUT
      pune_1 : Bool;
      pune_2 : Bool;
      pune_3 : Bool;
   END_VAR
BEGIN

REGION Network 1: daca e pornit, pune pentru forma1
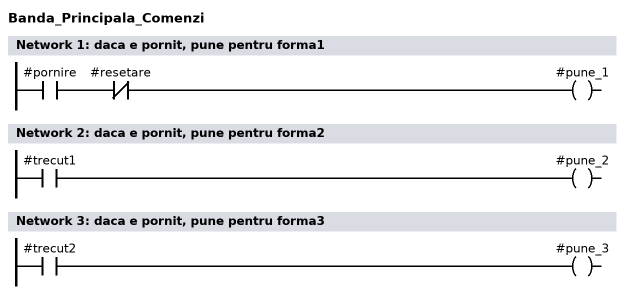
   RUNG wire#powerrail
      Contact( #pornire )
      I_Contact( #resetare )
      Coil( #pune_1 )
   END_RUNG
   // the same network as SCL:
   #pune_1 := #pornire AND NOT #resetare;
END_REGION

REGION Network 2: daca e pornit, pune pentru forma2
   RUNG wire#powerrail
      Contact( #trecut1 )
      Coil( #pune_2 )
   END_RUNG
   // the same network as SCL:
   #pune_2 := #trecut1;
END_REGION

REGION Network 3: daca e pornit, pune pentru forma3
   RUNG wire#powerrail
      Contact( #trecut2 )
      Coil( #pune_3 )
   END_RUNG
   // the same network as SCL:
   #pune_3 := #trecut2;
END_REGION
END_FUNCTION_BLOCK

FUNCTION_BLOCK "Banda_Principala_Simulare"   // FB5, LAD
{ S7_Optimized_Access := 'TRUE' }
VERSION : 0.1
   VAR_INPUT
      pune1 : Bool;
      pune2 : Bool;
      pune3 : Bool;
   END_VAR
   VAR_OUTPUT
      container_final : UInt;
      container_final_1 : UInt;
      container_final_2 : UInt;
      container_final_3 : UInt;
      trecut1 : Bool;
      trecut2 : Bool;
      trecut3 : Bool;
      resetare : Bool;
      alarma1 : Bool;
      alarma2 : Bool;
      alarma3 : Bool;
   END_VAR
   VAR_IN_OUT
      container1 : UInt;
      container2 : UInt;
      container3 : UInt;
      golire_container_final : Bool;
   END_VAR
   VAR
      timer_f1 : TON_TIME;
      timer_f2 : TON_TIME;
      timer_f3 : TON_TIME;
      re1 : Bool;
      reset_btn_golire : TON_TIME;
      timer_resetare : TON_TIME;
   END_VAR
   VAR_TEMP   // added for the SCL form of the ladder/FBD networks
      _w1 : Bool;
   END_VAR
BEGIN

REGION Network 1: daca poate pune pe 1, si containerulnu e pe 0, pune si continua
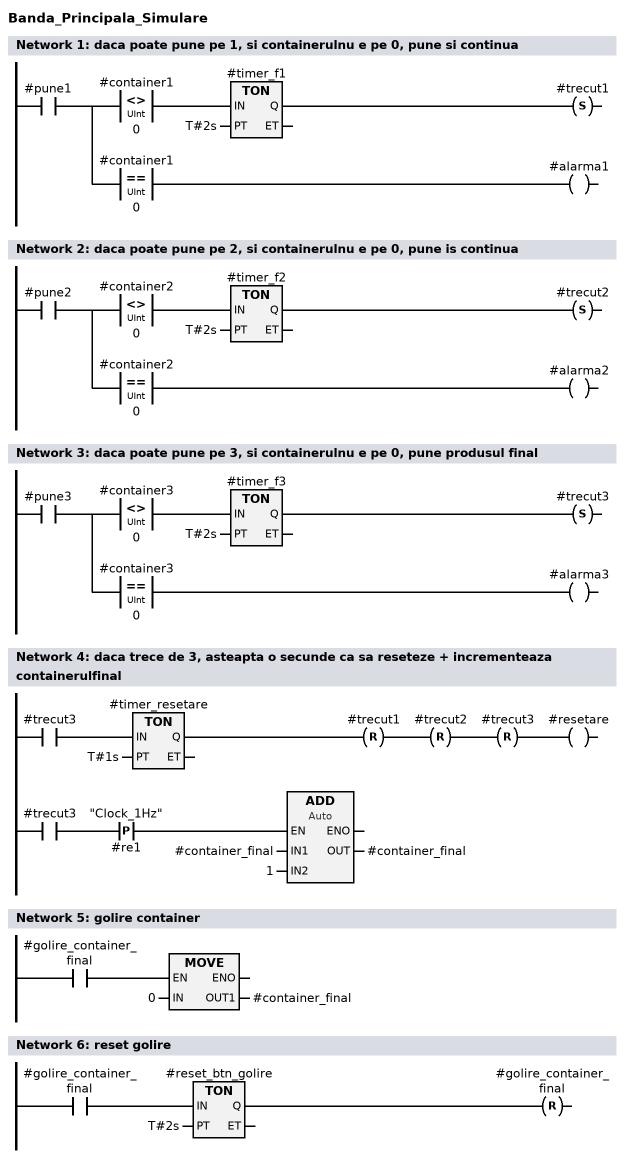
   #timer_f1(IN := #pune1 AND (#container1 <> 0), PT := T#2s);   // TON
   IF #timer_f1.Q THEN #trecut1 := TRUE; END_IF;
   #alarma1 := #pune1 AND (#container1 = 0);
END_REGION

REGION Network 2: daca poate pune pe 2, si containerulnu e pe 0, pune is continua
   #timer_f2(IN := #pune2 AND (#container2 <> 0), PT := T#2s);   // TON
   IF #timer_f2.Q THEN #trecut2 := TRUE; END_IF;
   #alarma2 := #pune2 AND (#container2 = 0);
END_REGION

REGION Network 3: daca poate pune pe 3, si containerulnu e pe 0, pune produsul final
   #timer_f3(IN := #pune3 AND (#container3 <> 0), PT := T#2s);   // TON
   IF #timer_f3.Q THEN #trecut3 := TRUE; END_IF;
   #alarma3 := #pune3 AND (#container3 = 0);
END_REGION

REGION Network 4: daca trece de 3, asteapta o secunde ca sa reseteze + incrementeaza containerulfinal
   #timer_resetare(IN := #trecut3, PT := T#1s);   // TON
   IF #timer_resetare.Q THEN
       #trecut1 := FALSE;
       #trecut2 := FALSE;
       #trecut3 := FALSE;
   END_IF;
   #resetare := #timer_resetare.Q;
   #_w1 := #trecut3 AND "Clock_1Hz" AND NOT #re1;   // rising edge of "Clock_1Hz"
   #re1 := "Clock_1Hz";
   IF #_w1 THEN #container_final := #container_final + 1; END_IF;
END_REGION

REGION Network 5: golire container
   RUNG wire#powerrail
      Contact( #golire_container_final )
      Move(in := 0, out1 => #container_final)
   END_RUNG
   // the same network as SCL:
   IF #golire_container_final THEN #container_final := 0; END_IF;
END_REGION

REGION Network 6: reset golire
   #reset_btn_golire(IN := #golire_container_final, PT := T#2s);   // TON
   IF #reset_btn_golire.Q THEN #golire_container_final := FALSE; END_IF;
END_REGION
END_FUNCTION_BLOCK

ORGANIZATION_BLOCK "Main"   // OB1, LAD, ProgramCycle
TITLE = "Main Program Sweep (Cycle)"
{ S7_Optimized_Access := 'TRUE' }
VERSION : 0.1
   VAR_INPUT
      Initial_Call : Bool;   // Initial call of this OB
      Remanence : Bool;   // =True, if remanent data are available
   END_VAR
BEGIN

REGION Network 1: banda1
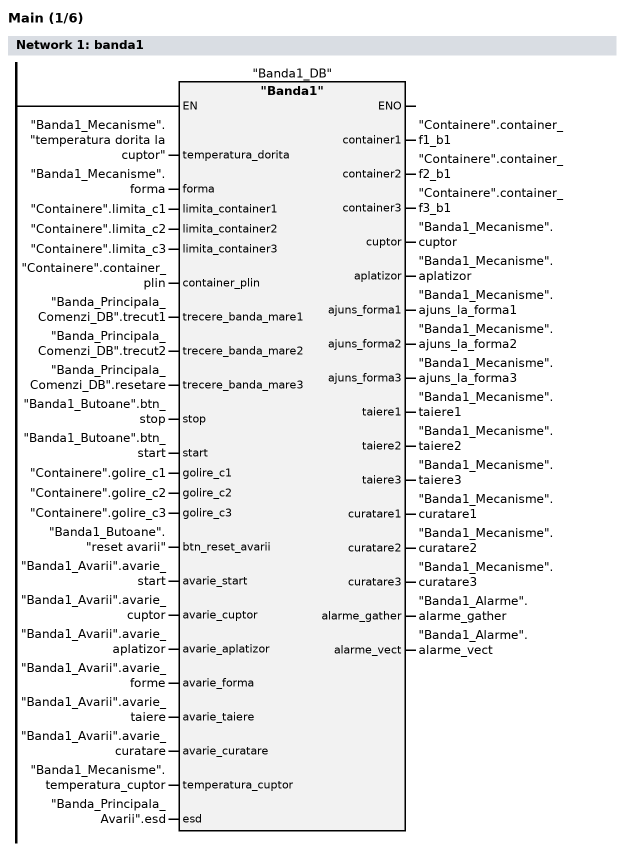
   RUNG wire#powerrail
      "Banda1_DB"(temperatura_dorita := "Banda1_Mecanisme"."temperatura dorita la cuptor", forma := "Banda1_Mecanisme".forma, limita_container1 := "Containere".limita_c1, limita_container2 := "Containere".limita_c2, limita_container3 := "Containere".limita_c3, container_plin := "Containere".container_plin, trecere_banda_mare1 := "Banda_Principala_Comenzi_DB".trecut1, trecere_banda_mare2 := "Banda_Principala_Comenzi_DB".trecut2, trecere_banda_mare3 := "Banda_Principala_Comenzi_DB".resetare, stop := "Banda1_Butoane".btn_stop, start := "Banda1_Butoane".btn_start, golire_c1 := "Containere".golire_c1, golire_c2 := "Containere".golire_c2, golire_c3 := "Containere".golire_c3, btn_reset_avarii := "Banda1_Butoane"."reset avarii", avarie_start := "Banda1_Avarii".avarie_start, avarie_cuptor := "Banda1_Avarii".avarie_cuptor, avarie_aplatizor := "Banda1_Avarii".avarie_aplatizor, avarie_forma := "Banda1_Avarii".avarie_forme, avarie_taiere := "Banda1_Avarii".avarie_taiere, avarie_curatare := "Banda1_Avarii".avarie_curatare, temperatura_cuptor := "Banda1_Mecanisme".temperatura_cuptor, esd := "Banda_Principala_Avarii".esd, container1 => "Containere".container_f1_b1, container2 => "Containere".container_f2_b1, container3 => "Containere".container_f3_b1, cuptor => "Banda1_Mecanisme".cuptor, aplatizor => "Banda1_Mecanisme".aplatizor, ajuns_forma1 => "Banda1_Mecanisme".ajuns_la_forma1, ajuns_forma2 => "Banda1_Mecanisme".ajuns_la_forma2, ajuns_forma3 => "Banda1_Mecanisme".ajuns_la_forma3, taiere1 => "Banda1_Mecanisme".taiere1, taiere2 => "Banda1_Mecanisme".taiere2, taiere3 => "Banda1_Mecanisme".taiere3, curatare1 => "Banda1_Mecanisme".curatare1, curatare2 => "Banda1_Mecanisme".curatare2, curatare3 => "Banda1_Mecanisme".curatare3, alarme_gather => "Banda1_Alarme".alarme_gather, alarme_vect => "Banda1_Alarme".alarme_vect)
   END_RUNG
   // the same network as SCL:
   "Banda1_DB"(temperatura_dorita := "Banda1_Mecanisme"."temperatura dorita la cuptor",   // "Banda1"
               forma := "Banda1_Mecanisme".forma,
               limita_container1 := "Containere".limita_c1,
               limita_container2 := "Containere".limita_c2,
               limita_container3 := "Containere".limita_c3,
               container_plin := "Containere".container_plin,
               trecere_banda_mare1 := "Banda_Principala_Comenzi_DB".trecut1,
               trecere_banda_mare2 := "Banda_Principala_Comenzi_DB".trecut2,
               trecere_banda_mare3 := "Banda_Principala_Comenzi_DB".resetare,
               stop := "Banda1_Butoane".btn_stop,
               start := "Banda1_Butoane".btn_start,
               golire_c1 := "Containere".golire_c1,
               golire_c2 := "Containere".golire_c2,
               golire_c3 := "Containere".golire_c3,
               btn_reset_avarii := "Banda1_Butoane"."reset avarii",
               avarie_start := "Banda1_Avarii".avarie_start,
               avarie_cuptor := "Banda1_Avarii".avarie_cuptor,
               avarie_aplatizor := "Banda1_Avarii".avarie_aplatizor,
               avarie_forma := "Banda1_Avarii".avarie_forme,
               avarie_taiere := "Banda1_Avarii".avarie_taiere,
               avarie_curatare := "Banda1_Avarii".avarie_curatare,
               temperatura_cuptor := "Banda1_Mecanisme".temperatura_cuptor,
               esd := "Banda_Principala_Avarii".esd,
               container1 => "Containere".container_f1_b1,
               container2 => "Containere".container_f2_b1,
               container3 => "Containere".container_f3_b1,
               cuptor => "Banda1_Mecanisme".cuptor,
               aplatizor => "Banda1_Mecanisme".aplatizor,
               ajuns_forma1 => "Banda1_Mecanisme".ajuns_la_forma1,
               ajuns_forma2 => "Banda1_Mecanisme".ajuns_la_forma2,
               ajuns_forma3 => "Banda1_Mecanisme".ajuns_la_forma3,
               taiere1 => "Banda1_Mecanisme".taiere1,
               taiere2 => "Banda1_Mecanisme".taiere2,
               taiere3 => "Banda1_Mecanisme".taiere3,
               curatare1 => "Banda1_Mecanisme".curatare1,
               curatare2 => "Banda1_Mecanisme".curatare2,
               curatare3 => "Banda1_Mecanisme".curatare3,
               alarme_gather => "Banda1_Alarme".alarme_gather,
               alarme_vect => "Banda1_Alarme".alarme_vect);
END_REGION

REGION Network 2: banda2
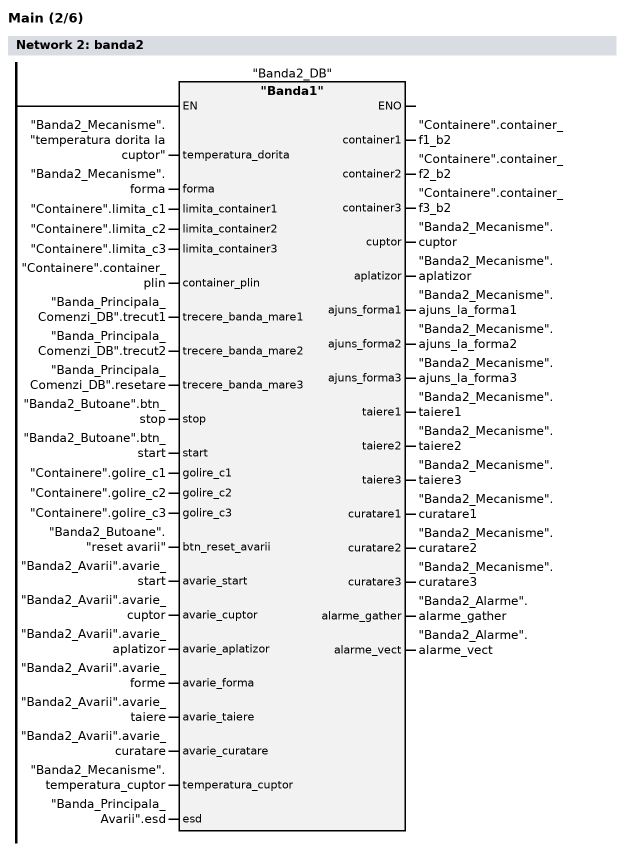
   RUNG wire#powerrail
      "Banda2_DB"(temperatura_dorita := "Banda2_Mecanisme"."temperatura dorita la cuptor", forma := "Banda2_Mecanisme".forma, limita_container1 := "Containere".limita_c1, limita_container2 := "Containere".limita_c2, limita_container3 := "Containere".limita_c3, container_plin := "Containere".container_plin, trecere_banda_mare1 := "Banda_Principala_Comenzi_DB".trecut1, trecere_banda_mare2 := "Banda_Principala_Comenzi_DB".trecut2, trecere_banda_mare3 := "Banda_Principala_Comenzi_DB".resetare, stop := "Banda2_Butoane".btn_stop, start := "Banda2_Butoane".btn_start, golire_c1 := "Containere".golire_c1, golire_c2 := "Containere".golire_c2, golire_c3 := "Containere".golire_c3, btn_reset_avarii := "Banda2_Butoane"."reset avarii", avarie_start := "Banda2_Avarii".avarie_start, avarie_cuptor := "Banda2_Avarii".avarie_cuptor, avarie_aplatizor := "Banda2_Avarii".avarie_aplatizor, avarie_forma := "Banda2_Avarii".avarie_forme, avarie_taiere := "Banda2_Avarii".avarie_taiere, avarie_curatare := "Banda2_Avarii".avarie_curatare, temperatura_cuptor := "Banda2_Mecanisme".temperatura_cuptor, esd := "Banda_Principala_Avarii".esd, container1 => "Containere".container_f1_b2, container2 => "Containere".container_f2_b2, container3 => "Containere".container_f3_b2, cuptor => "Banda2_Mecanisme".cuptor, aplatizor => "Banda2_Mecanisme".aplatizor, ajuns_forma1 => "Banda2_Mecanisme".ajuns_la_forma1, ajuns_forma2 => "Banda2_Mecanisme".ajuns_la_forma2, ajuns_forma3 => "Banda2_Mecanisme".ajuns_la_forma3, taiere1 => "Banda2_Mecanisme".taiere1, taiere2 => "Banda2_Mecanisme".taiere2, taiere3 => "Banda2_Mecanisme".taiere3, curatare1 => "Banda2_Mecanisme".curatare1, curatare2 => "Banda2_Mecanisme".curatare2, curatare3 => "Banda2_Mecanisme".curatare3, alarme_gather => "Banda2_Alarme".alarme_gather, alarme_vect => "Banda2_Alarme".alarme_vect)
   END_RUNG
   // the same network as SCL:
   "Banda2_DB"(temperatura_dorita := "Banda2_Mecanisme"."temperatura dorita la cuptor",   // "Banda1"
               forma := "Banda2_Mecanisme".forma,
               limita_container1 := "Containere".limita_c1,
               limita_container2 := "Containere".limita_c2,
               limita_container3 := "Containere".limita_c3,
               container_plin := "Containere".container_plin,
               trecere_banda_mare1 := "Banda_Principala_Comenzi_DB".trecut1,
               trecere_banda_mare2 := "Banda_Principala_Comenzi_DB".trecut2,
               trecere_banda_mare3 := "Banda_Principala_Comenzi_DB".resetare,
               stop := "Banda2_Butoane".btn_stop,
               start := "Banda2_Butoane".btn_start,
               golire_c1 := "Containere".golire_c1,
               golire_c2 := "Containere".golire_c2,
               golire_c3 := "Containere".golire_c3,
               btn_reset_avarii := "Banda2_Butoane"."reset avarii",
               avarie_start := "Banda2_Avarii".avarie_start,
               avarie_cuptor := "Banda2_Avarii".avarie_cuptor,
               avarie_aplatizor := "Banda2_Avarii".avarie_aplatizor,
               avarie_forma := "Banda2_Avarii".avarie_forme,
               avarie_taiere := "Banda2_Avarii".avarie_taiere,
               avarie_curatare := "Banda2_Avarii".avarie_curatare,
               temperatura_cuptor := "Banda2_Mecanisme".temperatura_cuptor,
               esd := "Banda_Principala_Avarii".esd,
               container1 => "Containere".container_f1_b2,
               container2 => "Containere".container_f2_b2,
               container3 => "Containere".container_f3_b2,
               cuptor => "Banda2_Mecanisme".cuptor,
               aplatizor => "Banda2_Mecanisme".aplatizor,
               ajuns_forma1 => "Banda2_Mecanisme".ajuns_la_forma1,
               ajuns_forma2 => "Banda2_Mecanisme".ajuns_la_forma2,
               ajuns_forma3 => "Banda2_Mecanisme".ajuns_la_forma3,
               taiere1 => "Banda2_Mecanisme".taiere1,
               taiere2 => "Banda2_Mecanisme".taiere2,
               taiere3 => "Banda2_Mecanisme".taiere3,
               curatare1 => "Banda2_Mecanisme".curatare1,
               curatare2 => "Banda2_Mecanisme".curatare2,
               curatare3 => "Banda2_Mecanisme".curatare3,
               alarme_gather => "Banda2_Alarme".alarme_gather,
               alarme_vect => "Banda2_Alarme".alarme_vect);
END_REGION

REGION Network 3: banda3
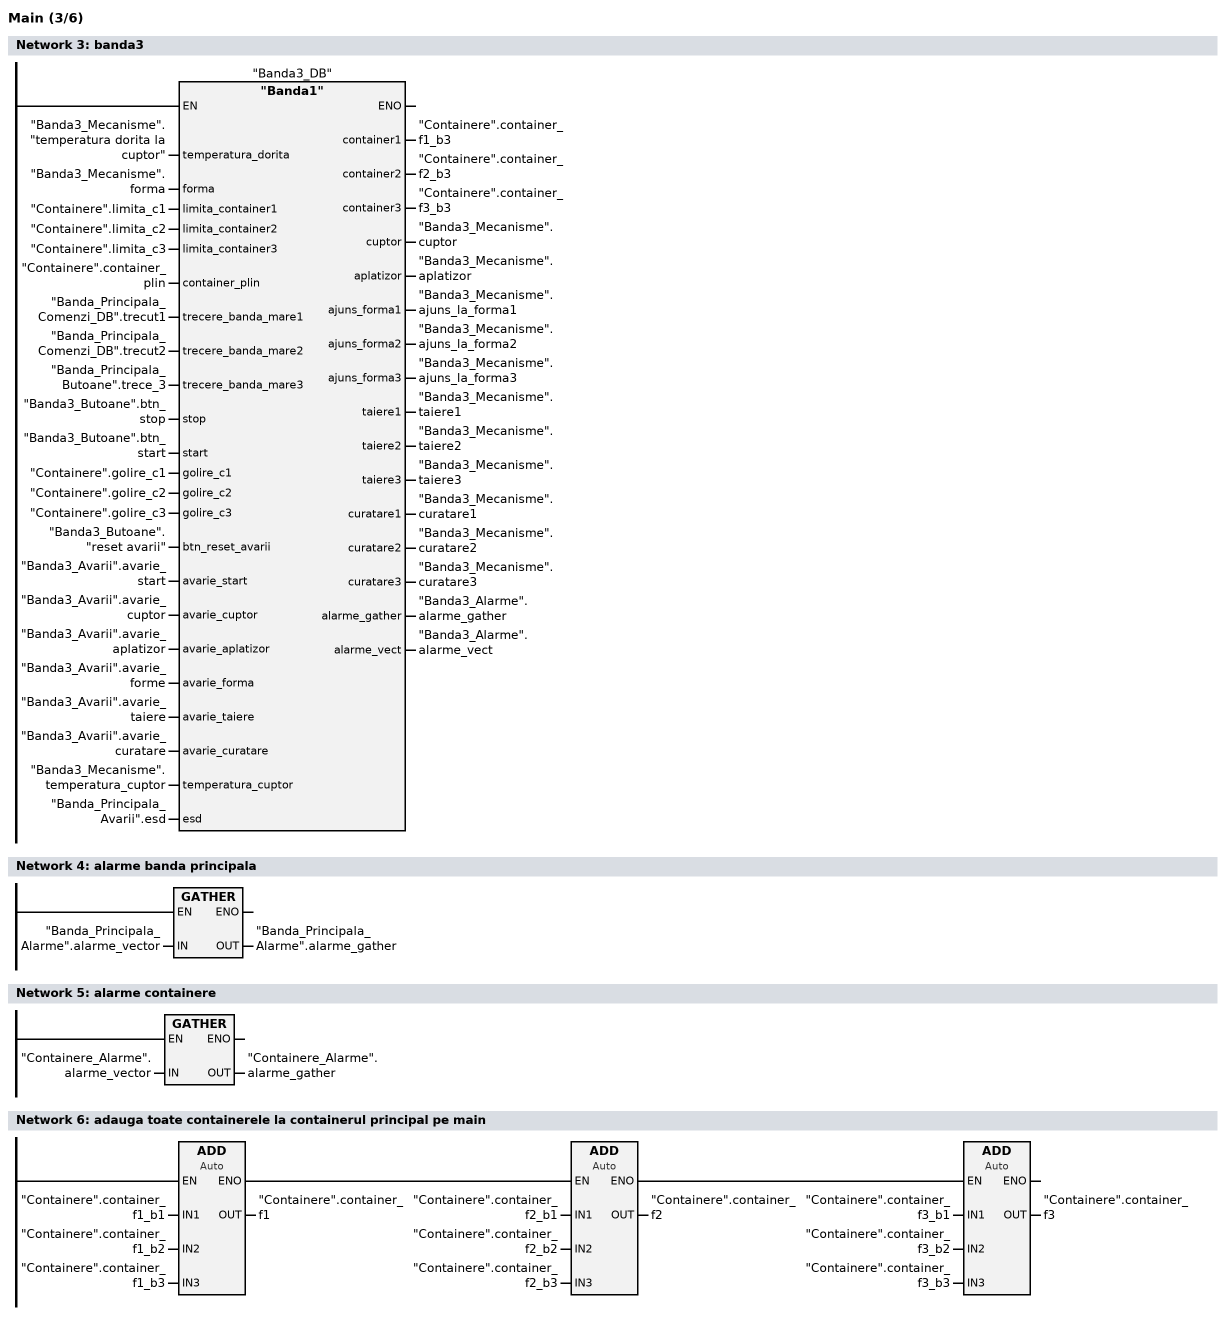
   RUNG wire#powerrail
      "Banda3_DB"(temperatura_dorita := "Banda3_Mecanisme"."temperatura dorita la cuptor", forma := "Banda3_Mecanisme".forma, limita_container1 := "Containere".limita_c1, limita_container2 := "Containere".limita_c2, limita_container3 := "Containere".limita_c3, container_plin := "Containere".container_plin, trecere_banda_mare1 := "Banda_Principala_Comenzi_DB".trecut1, trecere_banda_mare2 := "Banda_Principala_Comenzi_DB".trecut2, trecere_banda_mare3 := "Banda_Principala_Butoane".trece_3, stop := "Banda3_Butoane".btn_stop, start := "Banda3_Butoane".btn_start, golire_c1 := "Containere".golire_c1, golire_c2 := "Containere".golire_c2, golire_c3 := "Containere".golire_c3, btn_reset_avarii := "Banda3_Butoane"."reset avarii", avarie_start := "Banda3_Avarii".avarie_start, avarie_cuptor := "Banda3_Avarii".avarie_cuptor, avarie_aplatizor := "Banda3_Avarii".avarie_aplatizor, avarie_forma := "Banda3_Avarii".avarie_forme, avarie_taiere := "Banda3_Avarii".avarie_taiere, avarie_curatare := "Banda3_Avarii".avarie_curatare, temperatura_cuptor := "Banda3_Mecanisme".temperatura_cuptor, esd := "Banda_Principala_Avarii".esd, container1 => "Containere".container_f1_b3, container2 => "Containere".container_f2_b3, container3 => "Containere".container_f3_b3, cuptor => "Banda3_Mecanisme".cuptor, aplatizor => "Banda3_Mecanisme".aplatizor, ajuns_forma1 => "Banda3_Mecanisme".ajuns_la_forma1, ajuns_forma2 => "Banda3_Mecanisme".ajuns_la_forma2, ajuns_forma3 => "Banda3_Mecanisme".ajuns_la_forma3, taiere1 => "Banda3_Mecanisme".taiere1, taiere2 => "Banda3_Mecanisme".taiere2, taiere3 => "Banda3_Mecanisme".taiere3, curatare1 => "Banda3_Mecanisme".curatare1, curatare2 => "Banda3_Mecanisme".curatare2, curatare3 => "Banda3_Mecanisme".curatare3, alarme_gather => "Banda3_Alarme".alarme_gather, alarme_vect => "Banda3_Alarme".alarme_vect)
   END_RUNG
   // the same network as SCL:
   "Banda3_DB"(temperatura_dorita := "Banda3_Mecanisme"."temperatura dorita la cuptor",   // "Banda1"
               forma := "Banda3_Mecanisme".forma,
               limita_container1 := "Containere".limita_c1,
               limita_container2 := "Containere".limita_c2,
               limita_container3 := "Containere".limita_c3,
               container_plin := "Containere".container_plin,
               trecere_banda_mare1 := "Banda_Principala_Comenzi_DB".trecut1,
               trecere_banda_mare2 := "Banda_Principala_Comenzi_DB".trecut2,
               trecere_banda_mare3 := "Banda_Principala_Butoane".trece_3,
               stop := "Banda3_Butoane".btn_stop,
               start := "Banda3_Butoane".btn_start,
               golire_c1 := "Containere".golire_c1,
               golire_c2 := "Containere".golire_c2,
               golire_c3 := "Containere".golire_c3,
               btn_reset_avarii := "Banda3_Butoane"."reset avarii",
               avarie_start := "Banda3_Avarii".avarie_start,
               avarie_cuptor := "Banda3_Avarii".avarie_cuptor,
               avarie_aplatizor := "Banda3_Avarii".avarie_aplatizor,
               avarie_forma := "Banda3_Avarii".avarie_forme,
               avarie_taiere := "Banda3_Avarii".avarie_taiere,
               avarie_curatare := "Banda3_Avarii".avarie_curatare,
               temperatura_cuptor := "Banda3_Mecanisme".temperatura_cuptor,
               esd := "Banda_Principala_Avarii".esd,
               container1 => "Containere".container_f1_b3,
               container2 => "Containere".container_f2_b3,
               container3 => "Containere".container_f3_b3,
               cuptor => "Banda3_Mecanisme".cuptor,
               aplatizor => "Banda3_Mecanisme".aplatizor,
               ajuns_forma1 => "Banda3_Mecanisme".ajuns_la_forma1,
               ajuns_forma2 => "Banda3_Mecanisme".ajuns_la_forma2,
               ajuns_forma3 => "Banda3_Mecanisme".ajuns_la_forma3,
               taiere1 => "Banda3_Mecanisme".taiere1,
               taiere2 => "Banda3_Mecanisme".taiere2,
               taiere3 => "Banda3_Mecanisme".taiere3,
               curatare1 => "Banda3_Mecanisme".curatare1,
               curatare2 => "Banda3_Mecanisme".curatare2,
               curatare3 => "Banda3_Mecanisme".curatare3,
               alarme_gather => "Banda3_Alarme".alarme_gather,
               alarme_vect => "Banda3_Alarme".alarme_vect);
END_REGION

REGION Network 4: alarme banda principala
   GATHER(IN := "Banda_Principala_Alarme".alarme_vector, OUT => "Banda_Principala_Alarme".alarme_gather);
END_REGION

REGION Network 5: alarme containere
   GATHER(IN := "Containere_Alarme".alarme_vector, OUT => "Containere_Alarme".alarme_gather);
END_REGION

REGION Network 6: adauga toate containerele la containerul principal pe main
   RUNG wire#powerrail
      Add(in1 := "Containere".container_f1_b1, in2 := "Containere".container_f1_b2, in3 := "Containere".container_f1_b3, out => "Containere".container_f1)
      Add(in1 := "Containere".container_f2_b1, in2 := "Containere".container_f2_b2, in3 := "Containere".container_f2_b3, out => "Containere".container_f2)
      Add(in1 := "Containere".container_f3_b1, in2 := "Containere".container_f3_b2, in3 := "Containere".container_f3_b3, out => "Containere".container_f3)
   END_RUNG
   // the same network as SCL:
   "Containere".container_f1 := "Containere".container_f1_b1 + "Containere".container_f1_b2 + "Containere".container_f1_b3;
   "Containere".container_f2 := "Containere".container_f2_b1 + "Containere".container_f2_b2 + "Containere".container_f2_b3;
   "Containere".container_f3 := "Containere".container_f3_b1 + "Containere".container_f3_b2 + "Containere".container_f3_b3;
END_REGION

REGION Network 7: seteaza ca unul dincontainere e plin
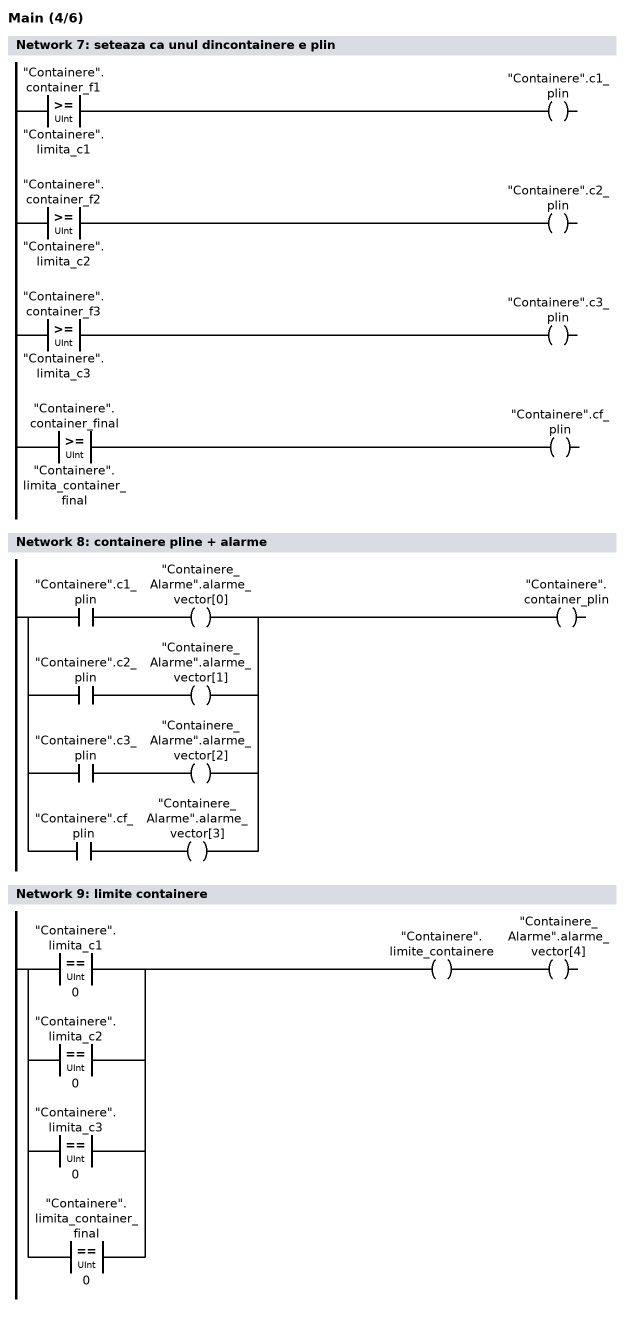
   RUNG wire#powerrail
      { S7_Templates := "SrcType := UInt" } GE_Contact(in1 := "Containere".container_f1, in2 := "Containere".limita_c1)
      Coil( "Containere".c1_plin )
   END_RUNG
   RUNG wire#powerrail
      { S7_Templates := "SrcType := UInt" } GE_Contact(in1 := "Containere".container_f2, in2 := "Containere".limita_c2)
      Coil( "Containere".c2_plin )
   END_RUNG
   RUNG wire#powerrail
      { S7_Templates := "SrcType := UInt" } GE_Contact(in1 := "Containere".container_f3, in2 := "Containere".limita_c3)
      Coil( "Containere".c3_plin )
   END_RUNG
   RUNG wire#powerrail
      { S7_Templates := "SrcType := UInt" } GE_Contact(in1 := "Containere".container_final, in2 := "Containere".limita_container_final)
      Coil( "Containere".cf_plin )
   END_RUNG
   // the same network as SCL:
   "Containere".c1_plin := "Containere".container_f1 >= "Containere".limita_c1;
   "Containere".c2_plin := "Containere".container_f2 >= "Containere".limita_c2;
   "Containere".c3_plin := "Containere".container_f3 >= "Containere".limita_c3;
   "Containere".cf_plin := "Containere".container_final >= "Containere".limita_container_final;
END_REGION

REGION Network 8: containere pline + alarme
   RUNG wire#powerrail
      Contact( "Containere".c1_plin )
      Coil( "Containere_Alarme".alarme_vector[0] )
      wire#w1
      Coil( "Containere".container_plin )
   END_RUNG
   RUNG wire#powerrail
      Contact( "Containere".c2_plin )
      Coil( "Containere_Alarme".alarme_vector[1] )
   END_RUNG wire#w1
   RUNG wire#powerrail
      Contact( "Containere".c3_plin )
      Coil( "Containere_Alarme".alarme_vector[2] )
   END_RUNG wire#w1
   RUNG wire#powerrail
      Contact( "Containere".cf_plin )
      Coil( "Containere_Alarme".alarme_vector[3] )
   END_RUNG wire#w1
   // the same network as SCL:
   "Containere_Alarme".alarme_vector[0] := "Containere".c1_plin;
   "Containere_Alarme".alarme_vector[1] := "Containere".c2_plin;
   "Containere_Alarme".alarme_vector[2] := "Containere".c3_plin;
   "Containere_Alarme".alarme_vector[3] := "Containere".cf_plin;
   "Containere".container_plin := "Containere".c1_plin OR "Containere".c2_plin OR "Containere".c3_plin OR "Containere".cf_plin;
END_REGION

REGION Network 9: limite containere
   RUNG wire#powerrail
      { S7_Templates := "SrcType := UInt" } EQ_Contact(in1 := "Containere".limita_c1, in2 := 0)
      wire#w1
      Coil( "Containere".limite_containere )
      Coil( "Containere_Alarme".alarme_vector[4] )
   END_RUNG
   RUNG wire#powerrail
      { S7_Templates := "SrcType := UInt" } EQ_Contact(in1 := "Containere".limita_c2, in2 := 0)
   END_RUNG wire#w1
   RUNG wire#powerrail
      { S7_Templates := "SrcType := UInt" } EQ_Contact(in1 := "Containere".limita_c3, in2 := 0)
   END_RUNG wire#w1
   RUNG wire#powerrail
      { S7_Templates := "SrcType := UInt" } EQ_Contact(in1 := "Containere".limita_container_final, in2 := 0)
   END_RUNG wire#w1
   // the same network as SCL:
   "Containere".limite_containere := ("Containere".limita_c1 = 0) OR ("Containere".limita_c2 = 0) OR ("Containere".limita_c3 = 0) OR ("Containere".limita_container_final = 0);
   "Containere_Alarme".alarme_vector[4] := "Containere".limite_containere;
END_REGION

REGION Network 10: pornire banda principala
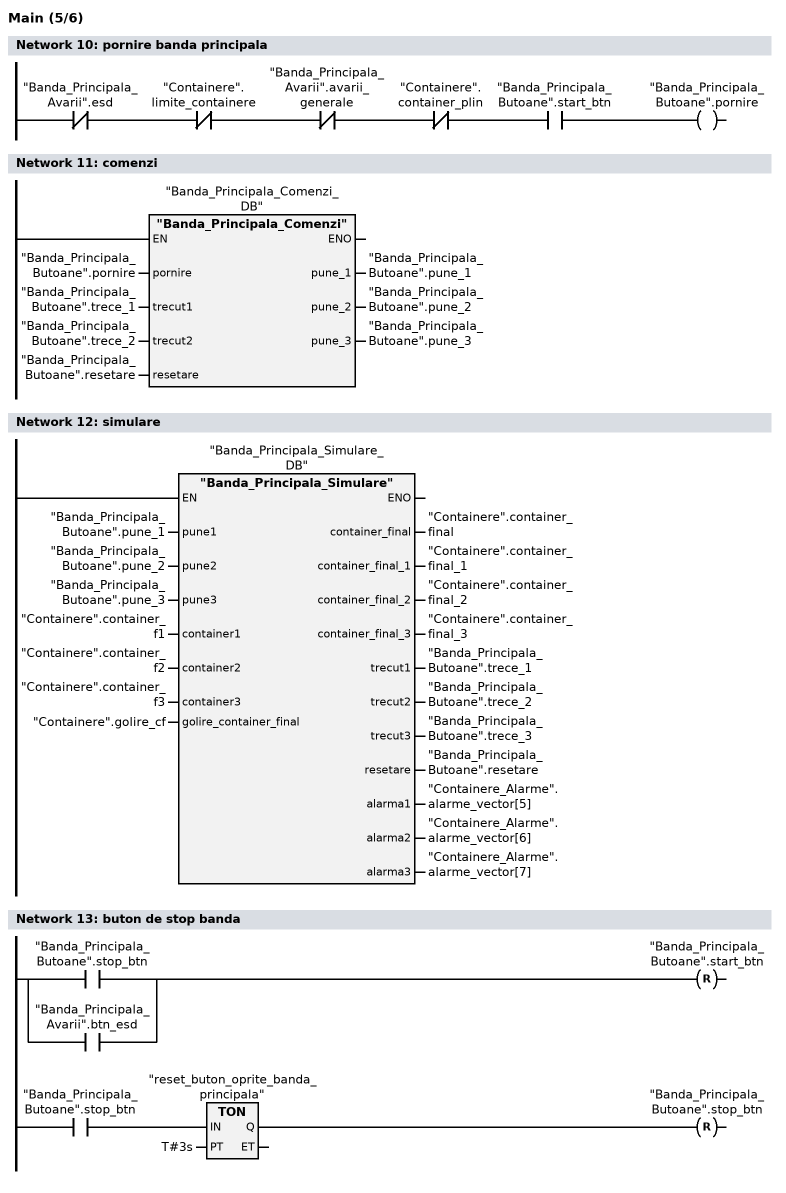
   RUNG wire#powerrail
      I_Contact( "Banda_Principala_Avarii".esd )
      I_Contact( "Containere".limite_containere )
      I_Contact( "Banda_Principala_Avarii".avarii_generale )
      I_Contact( "Containere".container_plin )
      Contact( "Banda_Principala_Butoane".start_btn )
      Coil( "Banda_Principala_Butoane".pornire )
   END_RUNG
   // the same network as SCL:
   "Banda_Principala_Butoane".pornire := NOT "Banda_Principala_Avarii".esd AND NOT "Containere".limite_containere AND NOT "Banda_Principala_Avarii".avarii_generale AND NOT "Containere".container_plin AND "Banda_Principala_Butoane".start_btn;
END_REGION

REGION Network 11: comenzi
   RUNG wire#powerrail
      "Banda_Principala_Comenzi_DB"(pornire := "Banda_Principala_Butoane".pornire, trecut1 := "Banda_Principala_Butoane".trece_1, trecut2 := "Banda_Principala_Butoane".trece_2, resetare := "Banda_Principala_Butoane".resetare, pune_1 => "Banda_Principala_Butoane".pune_1, pune_2 => "Banda_Principala_Butoane".pune_2, pune_3 => "Banda_Principala_Butoane".pune_3)
   END_RUNG
   // the same network as SCL:
   "Banda_Principala_Comenzi_DB"(pornire := "Banda_Principala_Butoane".pornire,   // "Banda_Principala_Comenzi"
                           trecut1 := "Banda_Principala_Butoane".trece_1,
                           trecut2 := "Banda_Principala_Butoane".trece_2,
                           resetare := "Banda_Principala_Butoane".resetare,
                           pune_1 => "Banda_Principala_Butoane".pune_1,
                           pune_2 => "Banda_Principala_Butoane".pune_2,
                           pune_3 => "Banda_Principala_Butoane".pune_3);
END_REGION

REGION Network 12: simulare
   RUNG wire#powerrail
      "Banda_Principala_Simulare_DB"(pune1 := "Banda_Principala_Butoane".pune_1, pune2 := "Banda_Principala_Butoane".pune_2, pune3 := "Banda_Principala_Butoane".pune_3, container1 := "Containere".container_f1, container2 := "Containere".container_f2, container3 := "Containere".container_f3, golire_container_final := "Containere".golire_cf, container_final => "Containere".container_final, container_final_1 => "Containere".container_final_1, container_final_2 => "Containere".container_final_2, container_final_3 => "Containere".container_final_3, trecut1 => "Banda_Principala_Butoane".trece_1, trecut2 => "Banda_Principala_Butoane".trece_2, trecut3 => "Banda_Principala_Butoane".trece_3, resetare => "Banda_Principala_Butoane".resetare, alarma1 => "Containere_Alarme".alarme_vector[5], alarma2 => "Containere_Alarme".alarme_vector[6], alarma3 => "Containere_Alarme".alarme_vector[7])
   END_RUNG
   // the same network as SCL:
   "Banda_Principala_Simulare_DB"(pune1 := "Banda_Principala_Butoane".pune_1,   // "Banda_Principala_Simulare"
                           pune2 := "Banda_Principala_Butoane".pune_2,
                           pune3 := "Banda_Principala_Butoane".pune_3,
                           container1 := "Containere".container_f1,
                           container2 := "Containere".container_f2,
                           container3 := "Containere".container_f3,
                           golire_container_final := "Containere".golire_cf,
                           container_final => "Containere".container_final,
                           container_final_1 => "Containere".container_final_1,
                           container_final_2 => "Containere".container_final_2,
                           container_final_3 => "Containere".container_final_3,
                           trecut1 => "Banda_Principala_Butoane".trece_1,
                           trecut2 => "Banda_Principala_Butoane".trece_2,
                           trecut3 => "Banda_Principala_Butoane".trece_3,
                           resetare => "Banda_Principala_Butoane".resetare,
                           alarma1 => "Containere_Alarme".alarme_vector[5],
                           alarma2 => "Containere_Alarme".alarme_vector[6],
                           alarma3 => "Containere_Alarme".alarme_vector[7]);
END_REGION

REGION Network 13: buton de stop banda
   IF "Banda_Principala_Butoane".stop_btn OR "Banda_Principala_Avarii".btn_esd THEN
       "Banda_Principala_Butoane".start_btn := FALSE;
   END_IF;
   "reset_buton_oprite_banda_principala".TON(IN := "Banda_Principala_Butoane".stop_btn, PT := T#3s);
   IF "reset_buton_oprite_banda_principala".Q THEN "Banda_Principala_Butoane".stop_btn := FALSE; END_IF;
END_REGION

REGION Network 14: setare avarie generala
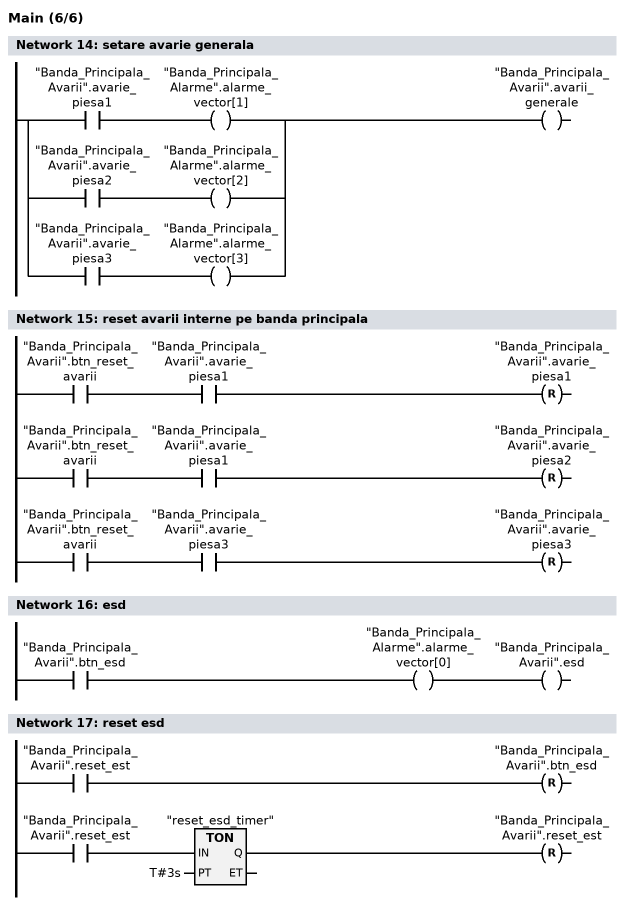
   RUNG wire#powerrail
      Contact( "Banda_Principala_Avarii".avarie_piesa1 )
      Coil( "Banda_Principala_Alarme".alarme_vector[1] )
      wire#w1
      Coil( "Banda_Principala_Avarii".avarii_generale )
   END_RUNG
   RUNG wire#powerrail
      Contact( "Banda_Principala_Avarii".avarie_piesa2 )
      Coil( "Banda_Principala_Alarme".alarme_vector[2] )
   END_RUNG wire#w1
   RUNG wire#powerrail
      Contact( "Banda_Principala_Avarii".avarie_piesa3 )
      Coil( "Banda_Principala_Alarme".alarme_vector[3] )
   END_RUNG wire#w1
   // the same network as SCL:
   "Banda_Principala_Alarme".alarme_vector[1] := "Banda_Principala_Avarii".avarie_piesa1;
   "Banda_Principala_Alarme".alarme_vector[2] := "Banda_Principala_Avarii".avarie_piesa2;
   "Banda_Principala_Alarme".alarme_vector[3] := "Banda_Principala_Avarii".avarie_piesa3;
   "Banda_Principala_Avarii".avarii_generale := "Banda_Principala_Avarii".avarie_piesa1 OR "Banda_Principala_Avarii".avarie_piesa2 OR "Banda_Principala_Avarii".avarie_piesa3;
END_REGION

REGION Network 15: reset avarii interne pe banda principala
   RUNG wire#powerrail
      Contact( "Banda_Principala_Avarii".btn_reset_avarii )
      Contact( "Banda_Principala_Avarii".avarie_piesa1 )
      R_Coil( "Banda_Principala_Avarii".avarie_piesa1 )
   END_RUNG
   RUNG wire#powerrail
      Contact( "Banda_Principala_Avarii".btn_reset_avarii )
      Contact( "Banda_Principala_Avarii".avarie_piesa1 )
      R_Coil( "Banda_Principala_Avarii".avarie_piesa2 )
   END_RUNG
   RUNG wire#powerrail
      Contact( "Banda_Principala_Avarii".btn_reset_avarii )
      Contact( "Banda_Principala_Avarii".avarie_piesa3 )
      R_Coil( "Banda_Principala_Avarii".avarie_piesa3 )
   END_RUNG
   // the same network as SCL:
   IF "Banda_Principala_Avarii".btn_reset_avarii AND "Banda_Principala_Avarii".avarie_piesa1 THEN
       "Banda_Principala_Avarii".avarie_piesa1 := FALSE;
   END_IF;
   IF "Banda_Principala_Avarii".btn_reset_avarii AND "Banda_Principala_Avarii".avarie_piesa1 THEN
       "Banda_Principala_Avarii".avarie_piesa2 := FALSE;
   END_IF;
   IF "Banda_Principala_Avarii".btn_reset_avarii AND "Banda_Principala_Avarii".avarie_piesa3 THEN
       "Banda_Principala_Avarii".avarie_piesa3 := FALSE;
   END_IF;
END_REGION

REGION Network 16: esd
   RUNG wire#powerrail
      Contact( "Banda_Principala_Avarii".btn_esd )
      Coil( "Banda_Principala_Alarme".alarme_vector[0] )
      Coil( "Banda_Principala_Avarii".esd )
   END_RUNG
   // the same network as SCL:
   "Banda_Principala_Alarme".alarme_vector[0] := "Banda_Principala_Avarii".btn_esd;
   "Banda_Principala_Avarii".esd := "Banda_Principala_Avarii".btn_esd;
END_REGION

REGION Network 17: reset esd
   IF "Banda_Principala_Avarii".reset_est THEN "Banda_Principala_Avarii".btn_esd := FALSE; END_IF;
   "reset_esd_timer".TON(IN := "Banda_Principala_Avarii".reset_est, PT := T#3s);
   IF "reset_esd_timer".Q THEN "Banda_Principala_Avarii".reset_est := FALSE; END_IF;
END_REGION
END_ORGANIZATION_BLOCK

(* ===== HMI "HMI_RT_1" =====
system functions are stored by id; their names below are inferred from use
connection "HMI_Connection_1": ETHERNET, SMART_S7_1500_OMS

HMI tags "Default tag table"
   "Tag_ScreenNumber" : UInt, internal
   "Banda_Principala_Butoane_start_btn" : Bool = PLC Banda_Principala_Butoane.start_btn, 1 s
   "Banda_Principala_Butoane_stop_btn" : Bool = PLC Banda_Principala_Butoane.stop_btn, 1 s
   "Banda_Principala_Avarii_btn_esd" : Bool = PLC Banda_Principala_Avarii.btn_esd, 1 s
   "Banda_Principala_Avarii_reset_est" : Bool = PLC Banda_Principala_Avarii.reset_est, 1 s
   "Banda_Principala_Avarii_esd" : Bool = PLC Banda_Principala_Avarii.esd, 1 s
   "Containere_container_f1" : UInt = PLC Containere.container_f1, 1 s
   "Containere_container_f2" : UInt = PLC Containere.container_f2, 1 s
   "Containere_container_f3" : UInt = PLC Containere.container_f3, 1 s
   "Containere_container_final" : UInt = PLC Containere.container_final, 1 s
   "Containere_limita_container_final" : UInt = PLC Containere.limita_container_final, 1 s
   "Banda_Principala_Butoane_trece_1" : Bool = PLC Banda_Principala_Butoane.trece_1, 1 s
   "Banda_Principala_Butoane_trece_2" : Bool = PLC Banda_Principala_Butoane.trece_2, 1 s
   "Banda_Principala_Butoane_trece_3" : Bool = PLC Banda_Principala_Butoane.trece_3, 1 s
   "Banda2_DB_start" : Bool = PLC Banda2_DB.start, 1 s
   "Banda2_DB_stop" : Bool = PLC Banda2_DB.stop, 1 s
   "Banda2_DB_temperatura_dorita" : Real = PLC Banda2_DB.temperatura_dorita, 1 s
   "Banda2_DB_temperatura_cuptor" : Real = PLC Banda2_DB.temperatura_cuptor, 1 s
   "Banda2_DB_cuptor" : Bool = PLC Banda2_DB.cuptor, 1 s
   "Banda2_DB_aplatizor" : Bool = PLC Banda2_DB.aplatizor, 1 s
   "Banda2_DB_forma" : UInt = PLC Banda2_DB.forma, 1 s
   "Containere_limita_c1" : UInt = PLC Containere.limita_c1, 1 s
   "Containere_limita_c2" : UInt = PLC Containere.limita_c2, 1 s
   "Containere_limita_c3" : UInt = PLC Containere.limita_c3, 1 s
   "Banda2_DB_ajuns_forma1" : Bool = PLC Banda2_DB.ajuns_forma1, 1 s
   "Banda2_DB_ajuns_forma2" : Bool = PLC Banda2_DB.ajuns_forma2, 1 s
   "Banda2_DB_ajuns_forma3" : Bool = PLC Banda2_DB.ajuns_forma3, 1 s
   "Banda2_DB_taiere1" : Bool = PLC Banda2_DB.taiere1, 1 s
   "Banda2_DB_taiere2" : Bool = PLC Banda2_DB.taiere2, 1 s
   "Banda2_DB_taiere3" : Bool = PLC Banda2_DB.taiere3, 1 s
   "Banda2_DB_curatare1" : Bool = PLC Banda2_DB.curatare1, 1 s
   "Banda2_DB_curatare2" : Bool = PLC Banda2_DB.curatare2, 1 s
   "Banda2_DB_curatare3" : Bool = PLC Banda2_DB.curatare3, 1 s
   "Banda2_DB_container1" : UInt = PLC Banda2_DB.container1, 1 s
   "Banda2_DB_container2" : UInt = PLC Banda2_DB.container2, 1 s
   "Banda2_DB_container3" : UInt = PLC Banda2_DB.container3, 1 s
   "Banda2_DB_golire_c1" : Bool = PLC Banda2_DB.golire_c1, 1 s
   "Banda2_DB_golire_c2" : Bool = PLC Banda2_DB.golire_c2, 1 s
   "Banda2_DB_golire_c3" : Bool = PLC Banda2_DB.golire_c3, 1 s
   "Containere_golire_c1" : Bool = PLC Containere.golire_c1, 1 s
   "Containere_golire_c2" : Bool = PLC Containere.golire_c2, 1 s
   "Containere_golire_c3" : Bool = PLC Containere.golire_c3, 1 s
   "Containere_golire_cf" : Bool = PLC Containere.golire_cf, 1 s
   "Banda3_DB_start" : Bool = PLC Banda3_DB.start, 1 s
   "Banda3_DB_stop" : Bool = PLC Banda3_DB.stop, 1 s
   "Banda3_DB_cuptor" : Bool = PLC Banda3_DB.cuptor, 1 s
   "Banda3_DB_temperatura_cuptor" : Real = PLC Banda3_DB.temperatura_cuptor, 1 s
   "Banda3_DB_aplatizor" : Bool = PLC Banda3_DB.aplatizor, 1 s
   "Banda3_DB_forma" : UInt = PLC Banda3_DB.forma, 1 s
   "Banda3_DB_ajuns_forma1" : Bool = PLC Banda3_DB.ajuns_forma1, 1 s
   "Banda3_DB_ajuns_forma2" : Bool = PLC Banda3_DB.ajuns_forma2, 1 s
   "Banda3_DB_ajuns_forma3" : Bool = PLC Banda3_DB.ajuns_forma3, 1 s
   "Banda3_DB_taiere1" : Bool = PLC Banda3_DB.taiere1, 1 s
   "Banda3_DB_taiere2" : Bool = PLC Banda3_DB.taiere2, 1 s
   "Banda3_DB_taiere3" : Bool = PLC Banda3_DB.taiere3, 1 s
   "Banda3_DB_curatare1" : Bool = PLC Banda3_DB.curatare1, 1 s
   "Banda3_DB_curatare2" : Bool = PLC Banda3_DB.curatare2, 1 s
   "Banda3_DB_curatare3" : Bool = PLC Banda3_DB.curatare3, 1 s
   "Banda3_DB_container1" : UInt = PLC Banda3_DB.container1, 1 s
   "Banda3_DB_container2" : UInt = PLC Banda3_DB.container2, 1 s
   "Banda3_DB_container3" : UInt = PLC Banda3_DB.container3, 1 s
   "Banda3_DB_golire_c1" : Bool = PLC Banda3_DB.golire_c1, 1 s
   "Banda3_DB_golire_c2" : Bool = PLC Banda3_DB.golire_c2, 1 s
   "Banda3_DB_golire_c3" : Bool = PLC Banda3_DB.golire_c3, 1 s
   "Banda3_DB_temperatura_dorita" : Real = PLC Banda3_DB.temperatura_dorita, 1 s
   "Banda1_DB_start" : Bool = PLC Banda1_DB.start, 1 s
   "Banda1_DB_stop" : Bool = PLC Banda1_DB.stop, 1 s
   "Banda1_DB_golire_c1" : Bool = PLC Banda1_DB.golire_c1, 1 s
   "Banda1_DB_golire_c2" : Bool = PLC Banda1_DB.golire_c2, 1 s
   "Banda1_DB_golire_c3" : Bool = PLC Banda1_DB.golire_c3, 1 s
   "Banda1_DB_forma" : UInt = PLC Banda1_DB.forma, 1 s
   "Banda1_DB_aplatizor" : Bool = PLC Banda1_DB.aplatizor, 1 s
   "Banda1_DB_cuptor" : Bool = PLC Banda1_DB.cuptor, 1 s
   "Banda1_DB_temperatura_cuptor" : Real = PLC Banda1_DB.temperatura_cuptor, 1 s
   "Banda1_DB_temperatura_dorita" : Real = PLC Banda1_DB.temperatura_dorita, 1 s
   "Banda1_DB_container1" : UInt = PLC Banda1_DB.container1, 1 s
   "Banda1_DB_container2" : UInt = PLC Banda1_DB.container2, 1 s
   "Banda1_DB_container3" : UInt = PLC Banda1_DB.container3, 1 s
   "Banda1_DB_ajuns_forma1" : Bool = PLC Banda1_DB.ajuns_forma1, 1 s
   "Banda1_DB_ajuns_forma2" : Bool = PLC Banda1_DB.ajuns_forma2, 1 s
   "Banda1_DB_ajuns_forma3" : Bool = PLC Banda1_DB.ajuns_forma3, 1 s
   "Banda1_DB_taiere1" : Bool = PLC Banda1_DB.taiere1, 1 s
   "Banda1_DB_taiere2" : Bool = PLC Banda1_DB.taiere2, 1 s
   "Banda1_DB_taiere3" : Bool = PLC Banda1_DB.taiere3, 1 s
   "Banda1_DB_curatare1" : Bool = PLC Banda1_DB.curatare1, 1 s
   "Banda1_DB_curatare2" : Bool = PLC Banda1_DB.curatare2, 1 s
   "Banda1_DB_curatare3" : Bool = PLC Banda1_DB.curatare3, 1 s
   "Banda1_DB_avarie_start" : Bool = PLC Banda1_DB.avarie_start, 1 s
   "Banda1_DB_avarie_cuptor" : Bool = PLC Banda1_DB.avarie_cuptor, 1 s
   "Banda1_DB_avarie_aplatizor" : Bool = PLC Banda1_DB.avarie_aplatizor, 1 s
   "Banda1_DB_avarie_forma" : Bool = PLC Banda1_DB.avarie_forma, 1 s
   "Banda1_DB_avarie_taiere" : Bool = PLC Banda1_DB.avarie_taiere, 1 s
   "Banda1_DB_avarie_curatare" : Bool = PLC Banda1_DB.avarie_curatare, 1 s
   "Banda1_DB_btn_reset_avarii" : Bool = PLC Banda1_DB.btn_reset_avarii, 1 s
   "Banda2_DB_avarie_start" : Bool = PLC Banda2_DB.avarie_start, 1 s
   "Banda2_DB_avarie_cuptor" : Bool = PLC Banda2_DB.avarie_cuptor, 1 s
   "Banda2_DB_avarie_aplatizor" : Bool = PLC Banda2_DB.avarie_aplatizor, 1 s
   "Banda2_DB_avarie_forma" : Bool = PLC Banda2_DB.avarie_forma, 1 s
   "Banda2_DB_avarie_taiere" : Bool = PLC Banda2_DB.avarie_taiere, 1 s
   "Banda2_DB_avarie_curatare" : Bool = PLC Banda2_DB.avarie_curatare, 1 s
   "Banda2_DB_btn_reset_avarii" : Bool = PLC Banda2_DB.btn_reset_avarii, 1 s
   "Banda3_DB_avarie_start" : Bool = PLC Banda3_DB.avarie_start, 1 s
   "Banda3_DB_avarie_cuptor" : Bool = PLC Banda3_DB.avarie_cuptor, 1 s
   "Banda3_DB_avarie_aplatizor" : Bool = PLC Banda3_DB.avarie_aplatizor, 1 s
   "Banda3_DB_avarie_forma" : Bool = PLC Banda3_DB.avarie_forma, 1 s
   "Banda3_DB_avarie_taiere" : Bool = PLC Banda3_DB.avarie_taiere, 1 s
   "Banda3_DB_avarie_curatare" : Bool = PLC Banda3_DB.avarie_curatare, 1 s
   "Banda3_DB_btn_reset_avarii" : Bool = PLC Banda3_DB.btn_reset_avarii, 1 s
   "Banda_Principala_Avarii_avarie_piesa1" : Bool = PLC Banda_Principala_Avarii.avarie_piesa1, 1 s
   "Banda_Principala_Avarii_avarie_piesa2" : Bool = PLC Banda_Principala_Avarii.avarie_piesa2, 1 s
   "Banda_Principala_Avarii_avarie_piesa3" : Bool = PLC Banda_Principala_Avarii.avarie_piesa3, 1 s
   "Banda_Principala_Avarii_btn_reset_avarii" : Bool = PLC Banda_Principala_Avarii.btn_reset_avarii, 1 s
   "Banda_Principala_Alarme_alarme_gather" : Word = PLC Banda_Principala_Alarme.alarme_gather, 1 s
   "Containere_Alarme_alarme_gather" : Word = PLC Containere_Alarme.alarme_gather, 1 s
   "Banda1_Alarme_alarme_gather" : Word = PLC Banda1_Alarme.alarme_gather, 1 s
   "Banda2_Alarme_alarme_gather" : Word = PLC Banda2_Alarme.alarme_gather, 1 s
   "Banda3_Alarme_alarme_gather" : Word = PLC Banda3_Alarme.alarme_gather, 1 s

discrete alarms
   1: 'ESD', class Errors, trigger "Banda_Principala_Alarme_alarme_gather" bit 0
   2: 'Piesa 1 defectata', class Errors, trigger "Banda_Principala_Alarme_alarme_gather" bit 1
   3: 'Piesa 2 defectata', class Errors, trigger "Banda_Principala_Alarme_alarme_gather" bit 2
   4: 'Piesa 3 defectata', class Errors, trigger "Banda_Principala_Alarme_alarme_gather" bit 3
   5: 'Nu mai sunt piese1', class Errors, trigger "Banda_Principala_Alarme_alarme_gather" bit 5
   6: 'Nu mai sunt piese2', class Errors, trigger "Banda_Principala_Alarme_alarme_gather" bit 6
   7: 'Nu mai sunt piese3', class Errors, trigger "Banda_Principala_Alarme_alarme_gather" bit 7
   8: 'Container 1 plin', class Errors, trigger "Containere_Alarme_alarme_gather" bit 0
   9: 'Container 2 plin', class Errors, trigger "Containere_Alarme_alarme_gather" bit 1
   10: 'Container 3 plin', class Errors, trigger "Containere_Alarme_alarme_gather" bit 2
   11: 'Container mare plin', class Errors, trigger "Containere_Alarme_alarme_gather" bit 3
   12: 'Limitele la containere nu sunt setate', class Errors, trigger "Containere_Alarme_alarme_gather" bit 4
   13: 'Banda1 avarie start', class Errors, trigger "Banda1_Alarme_alarme_gather" bit 1
   14: 'Banda1 avarie cuptor', class Errors, trigger "Banda1_Alarme_alarme_gather" bit 2
   15: 'Banda1 avarie aplatizor', class Errors, trigger "Banda1_Alarme_alarme_gather" bit 3
   16: 'Banda1 avarie forma', class Errors, trigger "Banda1_Alarme_alarme_gather" bit 4
   17: 'Banda1 avarie taiere', class Errors, trigger "Banda1_Alarme_alarme_gather" bit 5
   18: 'Banda1 avarie curatare', class Errors, trigger "Banda1_Alarme_alarme_gather" bit 6
   19: 'Banda2 avarie start', class Errors, trigger "Banda2_Alarme_alarme_gather" bit 1
   20: 'Banda2 avarie cuptor', class Errors, trigger "Banda2_Alarme_alarme_gather" bit 2
   21: 'Banda2 avarie aplatizor', class Errors, trigger "Banda2_Alarme_alarme_gather" bit 3
   22: 'Banda2 avarie forma', class Errors, trigger "Banda2_Alarme_alarme_gather" bit 4
   23: 'Banda2 avarie taiere', class Errors, trigger "Banda2_Alarme_alarme_gather" bit 5
   24: 'Banda2 avarie curatare', class Errors, trigger "Banda2_Alarme_alarme_gather" bit 6
   25: 'Banda3 avarie start', class Errors, trigger "Banda3_Alarme_alarme_gather" bit 1
   26: 'Banda3 avarie cuptor', class Errors, trigger "Banda3_Alarme_alarme_gather" bit 2
   27: 'Banda3 avarie aplatizor', class Errors, trigger "Banda3_Alarme_alarme_gather" bit 3
   28: 'Banda3 avarie forma', class Errors, trigger "Banda3_Alarme_alarme_gather" bit 4
   29: 'Banda3 avarie taiere', class Errors, trigger "Banda3_Alarme_alarme_gather" bit 5
   30: 'Banda3 avarie curatare', class Errors, trigger "Banda3_Alarme_alarme_gather" bit 6

text list "Forme": 0 'Forma1'; 1 'Forma2'; 2 'Forma3'

Template "Template_1" 800x480
   Button "Exit" at 722,440 size 55x39; TextOff 'Exit'; PictureOff "ExitRuntime_KTP900_Basic_PN_TR"; PictureOn "ExitRuntime_KTP900_Basic_PN_TR"
      on Release: StopRuntime(0)
   Button "Template_Button" at 622,440 size 55x39; TextOff 'Text'
   Button "Template_Button_1" at 522,440 size 55x39; TextOff 'Text'
   Button "Template_Button_2" at 422,440 size 55x39; TextOff 'Text'
   Button "Template_Button_3" at 322,440 size 55x39; TextOff 'Text'
   Button "Template_Button_4" at 222,440 size 55x39; TextOff 'Text'
   Button "Alarms" at 122,440 size 55x39; TextOff 'Alarms'; PictureOff "AlarmDisplay_KTP900_Basic_PN_TR"; PictureOn "AlarmDisplay_KTP900_Basic_PN_TR"
      on Release: function_ef3f5d25("Alarm window_1", -1)
   Button "Start screen" at 22,440 size 55x39; TextOff 'Start screen'; PictureOff "NavigateHome_KTP900_Basic_PN_TR"; PictureOn "NavigateHome_KTP900_Basic_PN_TR"
      on Release: ActivateScreen("Banda1", 0)
   SymbolicIOField "Symbolic_IO_Field_Screen" at 73,7 size 620x26; TextOff '0'; TextOn '1'; TextList "TextList_ScreenNames"
      ProcessValue <- "Tag_ScreenNumber"
      on Change: ActivateScreenByNumber("Tag_ScreenNumber", 0)
   DateTimeField "HmiScreenItemData" at 695,20 size 105x20
   DateTimeField "HmiScreenItemData_1" at 695,0 size 105x20
   GraphicView "Logo" at 0,0 size 71x40; Picture "Logo of HMI_1"

screen "Banda1" 800x480, template "Template_1"
   on GenerateScreen: SetTag("Tag_ScreenNumber", 1)
   TextField "Text field_1" at 319,37 size 93x32; Text 'Banda1'
   GraphicView "Graphic view_1" at 99,219 size 62x62; Picture "Graphic_1"
   GraphicView "Graphic view_6" at 197,168 size 105x59; Picture "Graphic_6"
      Visibility <- "Banda1_DB_aplatizor"
   Rectangle "Rectangle_2" at 323,299 size 108x20
      Appearance <- "Banda1_DB_ajuns_forma3"
   Rectangle "Rectangle_3" at 325,263 size 108x20
      Appearance <- "Banda1_DB_ajuns_forma2"
   Rectangle "Rectangle_4" at 326,226 size 108x20
      Appearance <- "Banda1_DB_ajuns_forma1"
   Rectangle "Rectangle_5" at 446,299 size 108x20
      Appearance <- "Banda1_DB_taiere3"
   Rectangle "Rectangle_6" at 447,262 size 108x20
      Appearance <- "Banda1_DB_taiere2"
   Rectangle "Rectangle_7" at 447,226 size 108x20
      Appearance <- "Banda1_DB_taiere1"
   Rectangle "Rectangle_8" at 566,299 size 108x20
      Appearance <- "Banda1_DB_curatare3"
   Rectangle "Rectangle_9" at 567,261 size 108x20
      Appearance <- "Banda1_DB_curatare2"
   Rectangle "Rectangle_10" at 567,224 size 108x20
      Appearance <- "Banda1_DB_curatare1"
   GraphicView "Graphic view_7" at 704,217 size 56x34; Picture "Graphic_9"
   Button "Button_1" at 14,145 size 42x32; TextOff 'Start'
      on Click: SetBit("Banda1_DB_start")
   SymbolicIOField "Symbolic I/O field_1" at 322,142 size 105x29; TextOff '0'; TextOn '1'; TextList "Forme"
      ProcessValue <- "Banda1_DB_forma"
   TextField "Text field_2" at 336,116 size 44x20; Text 'Forma'
   TextField "Text field_3" at 101,145 size 49x20; Text 'Cuptor'
   TextField "Text field_4" at 221,128 size 64x20; Text 'Aplatizor'
   TextField "Text field_5" at 478,143 size 45x20; Text 'Taiere'
   TextField "Text field_6" at 585,144 size 63x20; Text 'Curatare'
   TextField "Text field_7" at 696,145 size 68x20; Text 'Container'
   GraphicView "Graphic view_8" at 705,256 size 56x34; Picture "Graphic_9"
   GraphicView "Graphic view_9" at 705,295 size 56x34; Picture "Graphic_9"
   IOField "I/O field_1" at 159,352 size 48x32; FormatPattern 999
      ProcessValue <- "Banda1_DB_temperatura_dorita"
   IOField "I/O field_2" at 238,358 size 48x32; FormatPattern 999
      ProcessValue <- "Containere_limita_c2"
   IOField "I/O field_3" at 238,397 size 48x32; FormatPattern 999
      ProcessValue <- "Containere_limita_c3"
   IOField "I/O field_4" at 239,319 size 48x32; FormatPattern 999
      ProcessValue <- "Containere_limita_c1"
   TextField "Text field_8" at 137,328 size 89x20; Text 'Temperatura'
   TextField "Text field_9" at 202,293 size 117x20; Text 'Limite containere'
   Circle "Circle_2" at 108,178 size 31x31
      Appearance <- "Banda1_DB_cuptor"
   IOField "I/O field_5" at 711,223 size 42x23; FormatPattern 999
      ProcessValue <- "Banda1_DB_container1"
   IOField "I/O field_6" at 713,260 size 42x23; FormatPattern 999
      ProcessValue <- "Banda1_DB_container2"
   IOField "I/O field_7" at 712,299 size 42x23; FormatPattern 999
      ProcessValue <- "Banda1_DB_container3"
   Button "Button_4" at 548,380 size 32x32; TextOff 'C1'
      on Click: SetBit("Banda1_DB_golire_c1")
   Button "Button_5" at 631,379 size 32x32; TextOff 'C3'
      on Click: SetBit("Banda1_DB_golire_c3")
   Button "Button_6" at 590,380 size 32x32; TextOff 'C2'
      on Click: SetBit("Banda1_DB_golire_c2")
   TextField "Text field_10" at 549,355 size 116x20; Text 'Golire Containere'
   GraphicView "Graphic view_2" at 197,208 size 105x59; Picture "Graphic_6"
      Visibility <- "Banda1_DB_aplatizor"
   IOField "I/O field_8" at 102,107 size 48x32; FormatPattern 999
      ProcessValue <- "Banda1_DB_temperatura_cuptor"
   Button "Button_7" at 15,181 size 42x32; TextOff 'Stop'
      on Click: SetBit("Banda1_DB_stop")
   Button "Button_8" at 64,354 size 47x32; TextOff 'ESD'
      on Click: SetBit("Banda_Principala_Avarii_btn_esd")
   Button "Button_9" at 65,394 size 47x32; TextOff 'Reset'
      on Click: SetBit("Banda_Principala_Avarii_reset_est")
   Circle "Circle_3" at 71,314 size 31x31
      Appearance <- "Banda_Principala_Avarii_esd"

screen "Erori interne" 800x480
   TextField "Text field_1" at 310,4 size 152x32; Text 'Erori interne'
   Button "Button_1" at 53,139 size 57x25; TextOff 'Start'
      on Click: SetBit("Banda1_DB_avarie_start")
   Button "Button_2" at 53,183 size 57x25; TextOff 'Cuptor'
      on Click: SetBit("Banda1_DB_avarie_cuptor")
   Button "Button_3" at 53,227 size 57x25; TextOff 'Aplatizor'
      on Click: SetBit("Banda1_DB_avarie_aplatizor")
   Button "Button_4" at 53,271 size 57x25; TextOff 'Forme'
      on Click: SetBit("Banda1_DB_avarie_forma")
   Button "Button_5" at 53,315 size 57x25; TextOff 'Taiere'
      on Click: SetBit("Banda1_DB_avarie_taiere")
   Button "Button_6" at 53,359 size 57x25; TextOff 'Curatare'
      on Click: SetBit("Banda1_DB_avarie_curatare")
   Button "Button_7" at 119,241 size 57x42; TextOff 'Reset Avarii'
      on Click: SetBit("Banda1_DB_btn_reset_avarii")
   Circle "Circle_1" at 10,139 size 22x22
      Appearance <- "Banda1_DB_avarie_start"
   Circle "Circle_2" at 10,360 size 22x22
      Appearance <- "Banda1_DB_avarie_curatare"
   Circle "Circle_3" at 10,183 size 22x22
      Appearance <- "Banda1_DB_avarie_cuptor"
   Circle "Circle_4" at 10,227 size 22x22
      Appearance <- "Banda1_DB_avarie_aplatizor"
   Circle "Circle_5" at 10,271 size 22x22
      Appearance <- "Banda1_DB_avarie_forma"
   Circle "Circle_6" at 10,315 size 22x22
      Appearance <- "Banda1_DB_avarie_taiere"
   Button "Button_8" at 247,139 size 57x25; TextOff 'Start'
      on Click: SetBit("Banda2_DB_avarie_start")
   Button "Button_9" at 247,183 size 57x25; TextOff 'Cuptor'
      on Click: SetBit("Banda2_DB_avarie_cuptor")
   Button "Button_10" at 247,227 size 57x25; TextOff 'Aplatizor'
      on Click: SetBit("Banda2_DB_avarie_aplatizor")
   Button "Button_11" at 247,271 size 57x25; TextOff 'Forme'
      on Click: SetBit("Banda2_DB_avarie_forma")
   Button "Button_12" at 247,315 size 57x25; TextOff 'Taiere'
      on Click: SetBit("Banda2_DB_avarie_taiere")
   Button "Button_13" at 247,359 size 57x25; TextOff 'Curatare'
      on Click: SetBit("Banda2_DB_avarie_curatare")
   Button "Button_14" at 313,241 size 57x42; TextOff 'Reset Avarii'
      on Click: SetBit("Banda2_DB_btn_reset_avarii")
   Circle "Circle_7" at 204,139 size 22x22
      Appearance <- "Banda2_DB_avarie_start"
   Circle "Circle_8" at 204,360 size 22x22
      Appearance <- "Banda2_DB_avarie_curatare"
   Circle "Circle_9" at 204,183 size 22x22
      Appearance <- "Banda2_DB_avarie_cuptor"
   Circle "Circle_10" at 204,227 size 22x22
      Appearance <- "Banda2_DB_avarie_aplatizor"
   Circle "Circle_11" at 204,271 size 22x22
      Appearance <- "Banda2_DB_avarie_forma"
   Circle "Circle_12" at 204,315 size 22x22
      Appearance <- "Banda2_DB_avarie_taiere"
   Button "Button_15" at 445,139 size 57x25; TextOff 'Start'
      on Click: SetBit("Banda3_DB_avarie_start")
   Button "Button_16" at 445,183 size 57x25; TextOff 'Cuptor'
      on Click: SetBit("Banda3_DB_avarie_cuptor")
   Button "Button_17" at 445,227 size 57x25; TextOff 'Aplatizor'
      on Click: SetBit("Banda3_DB_avarie_aplatizor")
   Button "Button_18" at 445,271 size 57x25; TextOff 'Forme'
      on Click: SetBit("Banda3_DB_avarie_forma")
   Button "Button_19" at 445,315 size 57x25; TextOff 'Taiere'
      on Click: SetBit("Banda3_DB_avarie_taiere")
   Button "Button_20" at 445,359 size 57x25; TextOff 'Curatare'
      on Click: SetBit("Banda3_DB_avarie_curatare")
   Button "Button_21" at 511,241 size 57x42; TextOff 'Reset Avarii'
      on Click: SetBit("Banda3_DB_btn_reset_avarii")
   Circle "Circle_13" at 402,139 size 22x22
      Appearance <- "Banda3_DB_avarie_start"
   Circle "Circle_14" at 402,360 size 22x22
      Appearance <- "Banda3_DB_avarie_curatare"
   Circle "Circle_15" at 402,183 size 22x22
      Appearance <- "Banda3_DB_avarie_cuptor"
   Circle "Circle_16" at 402,227 size 22x22
      Appearance <- "Banda3_DB_avarie_aplatizor"
   Circle "Circle_17" at 402,271 size 22x22
      Appearance <- "Banda3_DB_avarie_forma"
   Circle "Circle_18" at 402,315 size 22x22
      Appearance <- "Banda3_DB_avarie_taiere"
   Button "Button_22" at 643,178 size 57x25; TextOff 'Piesa1'
      on Click: SetBit("Banda_Principala_Avarii_avarie_piesa1")
   Button "Button_24" at 643,227 size 57x25; TextOff 'Piesa2'
      on Click: SetBit("Banda_Principala_Avarii_avarie_piesa2")
   Button "Button_26" at 643,276 size 57x25; TextOff 'Piesa3'
      on Click: SetBit("Banda_Principala_Avarii_avarie_piesa3")
   Button "Button_28" at 643,337 size 57x42; TextOff 'Reset Avarii'
      on Click: SetBit("Banda_Principala_Avarii_btn_reset_avarii")
   Circle "Circle_19" at 600,178 size 22x22
      Appearance <- "Banda_Principala_Avarii_avarie_piesa1"
   Circle "Circle_22" at 600,227 size 22x22
      Appearance <- "Banda_Principala_Avarii_avarie_piesa2"
   Circle "Circle_24" at 600,276 size 22x22
      Appearance <- "Banda_Principala_Avarii_avarie_piesa3"
   TextField "Text field_2" at 60,79 size 70x25; Text 'Banda1'
   TextField "Text field_3" at 251,79 size 70x25; Text 'Banda2'
   TextField "Text field_4" at 450,78 size 70x25; Text 'Banda3'
   TextField "Text field_5" at 642,76 size 106x25; Text 'Banda Mare'

screen "Banda_principala" 800x480
   GraphicView "Graphic view_7" at 113,195 size 56x34; Picture "Graphic_9"
   TextField "Text field_7" at 105,123 size 68x20; Text 'Container'
   GraphicView "Graphic view_8" at 114,234 size 56x34; Picture "Graphic_9"
   GraphicView "Graphic view_9" at 114,273 size 56x34; Picture "Graphic_9"
   IOField "I/O field_5" at 120,201 size 42x23; FormatPattern 999
      ProcessValue <- "Containere_container_f1"
   IOField "I/O field_6" at 122,238 size 42x23; FormatPattern 999
      ProcessValue <- "Containere_container_f2"
   IOField "I/O field_7" at 121,277 size 42x23; FormatPattern 999
      ProcessValue <- "Containere_container_f3"
   Rectangle "Rectangle_3" at 209,241 size 108x20
      Appearance <- "Banda_Principala_Butoane_trece_1"
   Rectangle "Rectangle_6" at 331,240 size 108x20
      Appearance <- "Banda_Principala_Butoane_trece_2"
   Rectangle "Rectangle_9" at 451,239 size 108x20
      Appearance <- "Banda_Principala_Butoane_trece_3"
   TextField "Text field_1" at 237,201 size 47x20; Text 'Piesa1'
   TextField "Text field_2" at 479,199 size 47x20; Text 'Piesa3'
   TextField "Text field_3" at 360,199 size 47x20; Text 'Piesa2'
   GraphicView "Graphic view_1" at 597,219 size 131x67; Picture "Graphic_9"
   IOField "I/O field_1" at 626,241 size 73x29; FormatPattern 999
      ProcessValue <- "Containere_container_final"
   TextField "Text field_4" at 605,182 size 105x20; Text 'Container Mare'
   Button "Button_2" at 58,383 size 47x32; TextOff 'ESD'
      on Click: SetBit("Banda_Principala_Avarii_btn_esd")
   Button "Button_3" at 59,423 size 47x32; TextOff 'Reset'
      on Click: SetBit("Banda_Principala_Avarii_reset_est")
   Circle "Circle_1" at 65,343 size 31x31
      Appearance <- "Banda_Principala_Avarii_esd"
   Button "Button_1" at 23,52 size 42x32; TextOff 'Start'
      on Click: SetBit("Banda_Principala_Butoane_start_btn")
   Button "Button_7" at 24,88 size 42x32; TextOff 'Stop'
      on Click: SetBit("Banda_Principala_Butoane_stop_btn")
   IOField "I/O field_2" at 197,370 size 96x32; FormatPattern 999
      ProcessValue <- "Containere_limita_container_final"
   TextField "Text field_5" at 198,342 size 146x20; Text 'Limita container mare'
   Button "Button_4" at 450,375 size 32x32; TextOff 'C1'
      on Click: SetBit("Containere_golire_c1")
   Button "Button_5" at 533,374 size 32x32; TextOff 'C3'
      on Click: SetBit("Containere_golire_c3")
   Button "Button_6" at 492,375 size 32x32; TextOff 'C2'
      on Click: SetBit("Containere_golire_c2")
   TextField "Text field_10" at 451,350 size 116x20; Text 'Golire Containere'
   Button "Button_8" at 573,374 size 32x32; TextOff 'C.F.'
      on Click: SetBit("Containere_golire_cf")

screen "Banda2" 800x480
   TextField "Text field_1" at 319,37 size 93x32; Text 'Banda2'
   GraphicView "Graphic view_1" at 99,219 size 62x62; Picture "Graphic_1"
   GraphicView "Graphic view_6" at 197,168 size 105x59; Picture "Graphic_6"
      Visibility <- "Banda2_DB_aplatizor"
   Rectangle "Rectangle_2" at 323,299 size 108x20
      Appearance <- "Banda2_DB_ajuns_forma3"
   Rectangle "Rectangle_3" at 325,263 size 108x20
      Appearance <- "Banda2_DB_ajuns_forma2"
   Rectangle "Rectangle_4" at 326,226 size 108x20
      Appearance <- "Banda2_DB_ajuns_forma1"
   Rectangle "Rectangle_5" at 446,299 size 108x20
      Appearance <- "Banda2_DB_taiere3"
   Rectangle "Rectangle_6" at 447,262 size 108x20
      Appearance <- "Banda2_DB_taiere2"
   Rectangle "Rectangle_7" at 447,226 size 108x20
      Appearance <- "Banda2_DB_taiere1"
   Rectangle "Rectangle_8" at 566,299 size 108x20
      Appearance <- "Banda2_DB_curatare3"
   Rectangle "Rectangle_9" at 567,261 size 108x20
      Appearance <- "Banda2_DB_curatare2"
   Rectangle "Rectangle_10" at 567,224 size 108x20
      Appearance <- "Banda2_DB_curatare1"
   GraphicView "Graphic view_7" at 704,217 size 56x34; Picture "Graphic_9"
   Button "Button_1" at 14,145 size 42x32; TextOff 'Start'
      on Click: SetBit("Banda2_DB_start")
   SymbolicIOField "Symbolic I/O field_1" at 322,142 size 105x29; TextOn '1'; TextOff '0'; TextList "Forme"
      ProcessValue <- "Banda2_DB_forma"
   TextField "Text field_2" at 336,116 size 44x20; Text 'Forma'
   TextField "Text field_3" at 101,145 size 49x20; Text 'Cuptor'
   TextField "Text field_4" at 221,128 size 64x20; Text 'Aplatizor'
   TextField "Text field_5" at 478,143 size 45x20; Text 'Taiere'
   TextField "Text field_6" at 585,144 size 63x20; Text 'Curatare'
   TextField "Text field_7" at 696,145 size 68x20; Text 'Container'
   GraphicView "Graphic view_8" at 705,256 size 56x34; Picture "Graphic_9"
   GraphicView "Graphic view_9" at 705,295 size 56x34; Picture "Graphic_9"
   Button "Button_2" at 58,368 size 47x32; TextOff 'ESD'
      on Click: SetBit("Banda_Principala_Avarii_btn_esd")
   Button "Button_3" at 59,408 size 47x32; TextOff 'Reset'
      on Click: SetBit("Banda_Principala_Avarii_reset_est")
   Circle "Circle_1" at 65,328 size 31x31
      Appearance <- "Banda_Principala_Avarii_esd"
   IOField "I/O field_1" at 159,352 size 48x32; FormatPattern 999
      ProcessValue <- "Banda2_DB_temperatura_dorita"
   IOField "I/O field_2" at 238,358 size 48x32; FormatPattern 999
      ProcessValue <- "Containere_limita_c2"
   IOField "I/O field_3" at 238,397 size 48x32; FormatPattern 999
      ProcessValue <- "Containere_limita_c3"
   IOField "I/O field_4" at 239,319 size 48x32; FormatPattern 999
      ProcessValue <- "Containere_limita_c1"
   TextField "Text field_8" at 137,328 size 89x20; Text 'Temperatura'
   TextField "Text field_9" at 202,293 size 117x20; Text 'Limite containere'
   Circle "Circle_2" at 108,178 size 31x31
      Appearance <- "Banda2_DB_cuptor"
   IOField "I/O field_5" at 711,223 size 42x23; FormatPattern 999
      ProcessValue <- "Banda2_DB_container1"
   IOField "I/O field_6" at 713,260 size 42x23; FormatPattern 999
      ProcessValue <- "Banda2_DB_container2"
   IOField "I/O field_7" at 712,299 size 42x23; FormatPattern 999
      ProcessValue <- "Banda2_DB_container3"
   Button "Button_4" at 548,380 size 32x32; TextOff 'C1'
      on Click: SetBit("Banda2_DB_golire_c1")
   Button "Button_5" at 631,379 size 32x32; TextOff 'C3'
      on Click: SetBit("Banda2_DB_golire_c3")
   Button "Button_6" at 590,380 size 32x32; TextOff 'C2'
      on Click: SetBit("Banda2_DB_golire_c2")
   TextField "Text field_10" at 549,355 size 116x20; Text 'Golire Containere'
   GraphicView "Graphic view_2" at 197,208 size 105x59; Picture "Graphic_6"
      Visibility <- "Banda2_DB_aplatizor"
   IOField "I/O field_8" at 102,107 size 48x32; FormatPattern 999
      ProcessValue <- "Banda2_DB_temperatura_cuptor"
   Button "Button_7" at 15,181 size 42x32; TextOff 'Stop'
      on Click: SetBit("Banda2_DB_stop")

screen "Banda3" 800x480
   TextField "Text field_1" at 319,37 size 93x32; Text 'Banda3'
   GraphicView "Graphic view_1" at 99,219 size 62x62; Picture "Graphic_1"
   GraphicView "Graphic view_6" at 197,168 size 105x59; Picture "Graphic_6"
      Visibility <- "Banda3_DB_aplatizor"
   Rectangle "Rectangle_2" at 323,299 size 108x20
      Appearance <- "Banda3_DB_ajuns_forma3"
   Rectangle "Rectangle_3" at 325,263 size 108x20
      Appearance <- "Banda3_DB_ajuns_forma2"
   Rectangle "Rectangle_4" at 326,226 size 108x20
      Appearance <- "Banda3_DB_ajuns_forma1"
   Rectangle "Rectangle_5" at 446,299 size 108x20
      Appearance <- "Banda3_DB_taiere3"
   Rectangle "Rectangle_6" at 447,262 size 108x20
      Appearance <- "Banda3_DB_taiere2"
   Rectangle "Rectangle_7" at 447,226 size 108x20
      Appearance <- "Banda3_DB_taiere1"
   Rectangle "Rectangle_8" at 566,299 size 108x20
      Appearance <- "Banda3_DB_curatare3"
   Rectangle "Rectangle_9" at 567,261 size 108x20
      Appearance <- "Banda3_DB_curatare2"
   Rectangle "Rectangle_10" at 567,224 size 108x20
      Appearance <- "Banda3_DB_curatare1"
   GraphicView "Graphic view_7" at 704,217 size 56x34; Picture "Graphic_9"
   Button "Button_1" at 14,145 size 42x32; TextOff 'Start'
      on Click: SetBit("Banda3_DB_start")
   SymbolicIOField "Symbolic I/O field_1" at 322,142 size 105x29; TextOn '1'; TextOff '0'; TextList "Forme"
      ProcessValue <- "Banda3_DB_forma"
   TextField "Text field_2" at 336,116 size 44x20; Text 'Forma'
   TextField "Text field_3" at 101,145 size 49x20; Text 'Cuptor'
   TextField "Text field_4" at 221,128 size 64x20; Text 'Aplatizor'
   TextField "Text field_5" at 478,143 size 45x20; Text 'Taiere'
   TextField "Text field_6" at 585,144 size 63x20; Text 'Curatare'
   TextField "Text field_7" at 696,145 size 68x20; Text 'Container'
   GraphicView "Graphic view_8" at 705,256 size 56x34; Picture "Graphic_9"
   GraphicView "Graphic view_9" at 705,295 size 56x34; Picture "Graphic_9"
   IOField "I/O field_1" at 159,352 size 48x32; FormatPattern 999
      ProcessValue <- "Banda3_DB_temperatura_dorita"
   IOField "I/O field_2" at 238,358 size 48x32; FormatPattern 999
      ProcessValue <- "Containere_limita_c2"
   IOField "I/O field_3" at 238,397 size 48x32; FormatPattern 999
      ProcessValue <- "Containere_limita_c3"
   IOField "I/O field_4" at 239,319 size 48x32; FormatPattern 999
      ProcessValue <- "Containere_limita_c1"
   TextField "Text field_8" at 137,328 size 89x20; Text 'Temperatura'
   TextField "Text field_9" at 202,293 size 117x20; Text 'Limite containere'
   Circle "Circle_2" at 108,178 size 31x31
      Appearance <- "Banda3_DB_cuptor"
   IOField "I/O field_5" at 711,223 size 42x23; FormatPattern 999
      ProcessValue <- "Banda3_DB_container1"
   IOField "I/O field_6" at 713,260 size 42x23; FormatPattern 999
      ProcessValue <- "Banda3_DB_container2"
   IOField "I/O field_7" at 712,299 size 42x23; FormatPattern 999
      ProcessValue <- "Banda3_DB_container3"
   Button "Button_4" at 548,380 size 32x32; TextOff 'C1'
      on Click: SetBit("Banda3_DB_golire_c1")
   Button "Button_5" at 631,379 size 32x32; TextOff 'C3'
      on Click: SetBit("Banda3_DB_golire_c3")
   Button "Button_6" at 590,380 size 32x32; TextOff 'C2'
      on Click: SetBit("Banda3_DB_golire_c2")
   TextField "Text field_10" at 549,355 size 116x20; Text 'Golire Containere'
   GraphicView "Graphic view_2" at 197,208 size 105x59; Picture "Graphic_6"
      Visibility <- "Banda3_DB_aplatizor"
   IOField "I/O field_8" at 102,107 size 48x32; FormatPattern 999
      ProcessValue <- "Banda3_DB_temperatura_cuptor"
   Button "Button_7" at 15,181 size 42x32; TextOff 'Stop'
      on Click: SetBit("Banda3_DB_stop")
   Button "Button_8" at 61,365 size 47x32; TextOff 'ESD'
      on Click: SetBit("Banda_Principala_Avarii_btn_esd")
   Button "Button_9" at 62,405 size 47x32; TextOff 'Reset'
      on Click: SetBit("Banda_Principala_Avarii_reset_est")
   Circle "Circle_3" at 68,325 size 31x31
      Appearance <- "Banda_Principala_Avarii_esd"
*)